Yaskawa INFORM job: DPRINT3D13.JBI

/JOB
//NAME DPRINT3D13
//POS
///NPOS 947,0,0,0,0,0
///TOOL 9
///POSTYPE PULSE
///PULSE
C00000=36504,50728,-112236,78231,-119117,-87318,0
C00001=42210,46378,-124713,70675,-118736,-91580,0
C00002=39842,45351,-127762,72820,-116851,-92177,0
C00003=34258,49660,-115138,80114,-117255,-87892,0
C00004=35160,50071,-114017,79347,-117985,-87668,0
C00005=34925,50304,-113369,79663,-117991,-87456,0
C00006=35393,50528,-112763,79272,-118380,-87336,0
C00007=35576,50347,-113263,79025,-118376,-87500,0
C00008=36136,50038,-114124,78353,-118497,-87812,0
C00009=41210,45662,-126843,71472,-117684,-92067,0
C00010=42439,44983,-128954,69897,-117543,-92821,0
C00011=39332,48664,-118025,74580,-119242,-89315,0
C00012=41658,49917,-114566,72665,-121338,-88655,0
C00013=34878,50571,-112636,79801,-118117,-87241,0
C00014=33997,51512,-110060,80995,-118129,-86405,0
C00015=36100,49514,-115576,78205,-118155,-88224,0
C00016=40170,46391,-124628,72850,-117873,-91306,0
C00017=40171,46330,-124643,72860,-117898,-91281,0
C00018=33600,46215,-124852,79721,-114877,-90646,0
C00019=36393,47272,-121802,77159,-116891,-90027,0
C00020=36323,49924,-114301,78154,-118581,-87857,0
C00021=40982,46356,-124583,72010,-118271,-91361,0
C00022=39975,45915,-125877,72916,-117468,-91614,0
C00023=35360,49470,-115543,78969,-117787,-88102,0
C00024=36245,49887,-114404,78220,-118516,-87877,0
C00025=35630,50238,-113425,78963,-118392,-87525,0
C00026=36504,50672,-112251,78242,-119134,-87295,0
C00027=42210,46316,-124729,70686,-118763,-91556,0
C00028=39843,45287,-127778,72830,-116876,-92151,0
C00029=34259,49603,-115155,80124,-117272,-87868,0
C00030=35161,50014,-114032,79357,-118002,-87645,0
C00031=34925,50248,-113384,79673,-118008,-87433,0
C00032=35394,50472,-112778,79282,-118397,-87313,0
C00033=35576,50291,-113278,79035,-118393,-87477,0
C00034=36137,49982,-114139,78363,-118516,-87789,0
C00035=41210,45599,-126858,71483,-117710,-92041,0
C00036=42421,44928,-128939,69931,-117572,-92784,0
C00037=39332,48606,-118041,74591,-119264,-89291,0
C00038=41626,49842,-114632,72703,-121329,-88642,0
C00039=34879,50515,-112651,79811,-118134,-87218,0
C00040=34010,51443,-110113,80987,-118144,-86395,0
C00041=36100,49457,-115591,78215,-118173,-88200,0
C00042=40171,46330,-124643,72860,-117898,-91281,0
C00043=40171,46268,-124659,72871,-117922,-91256,0
C00044=33640,46167,-124827,79692,-114924,-90612,0
C00045=36394,47211,-121817,77168,-116912,-90002,0
C00046=36324,49868,-114316,78165,-118600,-87834,0
C00047=40982,46294,-124599,72020,-118295,-91336,0
C00048=39976,45852,-125893,72926,-117492,-91589,0
C00049=35360,49413,-115558,78979,-117805,-88078,0
C00050=36246,49830,-114419,78230,-118534,-87854,0
C00051=35631,50182,-113440,78973,-118409,-87502,0
C00052=36504,50617,-112266,78252,-119152,-87272,0
C00053=42211,46254,-124744,70697,-118789,-91531,0
C00054=39843,45223,-127794,72840,-116901,-92125,0
C00055=34259,49546,-115170,80133,-117290,-87845,0
C00056=35161,49958,-114047,79366,-118019,-87622,0
C00057=34926,50192,-113399,79682,-118025,-87410,0
C00058=35394,50417,-112793,79292,-118415,-87290,0
C00059=35577,50235,-113293,79045,-118410,-87454,0
C00060=36137,49925,-114154,78373,-118533,-87765,0
C00061=41211,45536,-126874,71493,-117736,-92016,0
C00062=42403,44874,-128924,69965,-117602,-92748,0
C00063=39333,48548,-118056,74602,-119286,-89268,0
C00064=41594,49766,-114699,72740,-121321,-88629,0
C00065=34879,50459,-112666,79821,-118152,-87195,0
C00066=34023,51374,-110166,80980,-118160,-86384,0
C00067=36101,49400,-115607,78225,-118192,-88177,0
C00068=40171,46268,-124659,72871,-117922,-91256,0
C00069=40172,46206,-124674,72881,-117946,-91231,0
C00070=33681,46119,-124803,79663,-114971,-90578,0
C00071=36394,47151,-121832,77178,-116932,-89977,0
C00072=36324,49811,-114331,78175,-118618,-87811,0
C00073=40982,46232,-124614,72031,-118321,-91312,0
C00074=39976,45790,-125908,72937,-117517,-91563,0
C00075=35361,49356,-115573,78988,-117823,-88054,0
C00076=36246,49773,-114434,78240,-118553,-87830,0
C00077=35631,50126,-113455,78983,-118427,-87479,0
C00078=36505,50561,-112281,78263,-119171,-87249,0
C00079=42211,46192,-124760,70708,-118815,-91506,0
C00080=39843,45159,-127810,72850,-116927,-92100,0
C00081=34259,49489,-115184,80143,-117307,-87821,0
C00082=35161,49901,-114062,79376,-118037,-87599,0
C00083=34926,50136,-113414,79692,-118042,-87386,0
C00084=35394,50361,-112807,79302,-118432,-87267,0
C00085=35577,50179,-113308,79056,-118429,-87431,0
C00086=36137,49869,-114169,78383,-118551,-87742,0
C00087=41211,45472,-126890,71503,-117762,-91991,0
C00088=42385,44819,-128910,69999,-117632,-92711,0
C00089=39333,48489,-118071,74612,-119308,-89244,0
C00090=41562,49691,-114766,72778,-121312,-88616,0
C00091=34879,50404,-112681,79830,-118168,-87172,0
C00092=34036,51306,-110219,80972,-118176,-86374,0
C00093=36101,49343,-115622,78235,-118210,-88153,0
C00094=40172,46206,-124674,72881,-117946,-91231,0
C00095=40172,46144,-124690,72892,-117970,-91206,0
C00096=33721,46071,-124778,79635,-115017,-90544,0
C00097=36394,47091,-121848,77188,-116953,-89953,0
C00098=36324,49755,-114346,78185,-118637,-87787,0
C00099=40983,46170,-124631,72041,-118346,-91287,0
C00100=39976,45727,-125924,72947,-117541,-91538,0
C00101=35361,49299,-115588,78998,-117841,-88031,0
C00102=36246,49717,-114449,78250,-118571,-87807,0
C00103=35631,50070,-113469,78993,-118445,-87456,0
C00104=36505,50505,-112296,78273,-119188,-87226,0
C00105=42212,46130,-124775,70718,-118841,-91482,0
C00106=39844,45095,-127825,72860,-116952,-92074,0
C00107=34260,49432,-115199,80152,-117324,-87797,0
C00108=35161,49845,-114077,79386,-118054,-87576,0
C00109=34926,50080,-113429,79702,-118060,-87363,0
C00110=35395,50305,-112822,79312,-118449,-87244,0
C00111=35577,50123,-113323,79066,-118446,-87408,0
C00112=36138,49813,-114184,78394,-118570,-87719,0
C00113=41212,45409,-126905,71514,-117787,-91966,0
C00114=42367,44764,-128895,70033,-117662,-92674,0
C00115=39333,48431,-118086,74623,-119328,-89220,0
C00116=41530,49615,-114832,72816,-121304,-88603,0
C00117=34880,50348,-112696,79840,-118185,-87149,0
C00118=34049,51237,-110272,80965,-118192,-86364,0
C00119=36101,49286,-115637,78245,-118230,-88129,0
C00120=40172,46144,-124690,72892,-117970,-91206,0
C00121=40173,46082,-124705,72902,-117995,-91181,0
C00122=33761,46023,-124752,79606,-115064,-90509,0
C00123=36395,47031,-121863,77198,-116974,-89928,0
C00124=36325,49699,-114361,78195,-118655,-87764,0
C00125=40983,46108,-124645,72052,-118370,-91262,0
C00126=39977,45665,-125939,72957,-117567,-91513,0
C00127=35361,49242,-115603,79008,-117859,-88007,0
C00128=36247,49661,-114464,78260,-118589,-87784,0
C00129=35632,50014,-113484,79003,-118462,-87433,0
C00130=36505,50450,-112310,78283,-119207,-87203,0
C00131=42212,46068,-124791,70729,-118866,-91457,0
C00132=39844,45031,-127841,72870,-116977,-92048,0
C00133=34260,49376,-115213,80162,-117341,-87773,0
C00134=35162,49789,-114092,79396,-118072,-87552,0
C00135=34927,50024,-113444,79712,-118077,-87340,0
C00136=35395,50249,-112837,79322,-118466,-87220,0
C00137=35578,50067,-113337,79076,-118463,-87385,0
C00138=36138,49756,-114199,78404,-118588,-87696,0
C00139=41212,45346,-126921,71524,-117814,-91940,0
C00140=42349,44709,-128880,70067,-117692,-92638,0
C00141=39334,48373,-118101,74634,-119350,-89196,0
C00142=41497,49539,-114898,72854,-121295,-88589,0
C00143=34880,50292,-112711,79850,-118202,-87125,0
C00144=34062,51168,-110325,80957,-118207,-86354,0
C00145=36102,49229,-115651,78255,-118248,-88106,0
C00146=40173,46082,-124705,72902,-117995,-91181,0
C00147=40173,46020,-124720,72913,-118019,-91156,0
C00148=33801,45976,-124727,79578,-115111,-90475,0
C00149=36395,46971,-121878,77207,-116993,-89903,0
C00150=36325,49642,-114375,78206,-118673,-87740,0
C00151=40984,46047,-124660,72063,-118395,-91237,0
C00152=39977,45602,-125955,72967,-117591,-91488,0
C00153=35362,49185,-115618,79018,-117877,-87984,0
C00154=36247,49604,-114478,78271,-118608,-87761,0
C00155=35632,49958,-113499,79013,-118480,-87410,0
C00156=36506,50394,-112325,78294,-119224,-87180,0
C00157=42212,46006,-124806,70740,-118893,-91433,0
C00158=39845,44968,-127856,72880,-117002,-92022,0
C00159=34260,49319,-115228,80171,-117359,-87750,0
C00160=35162,49733,-114106,79406,-118090,-87529,0
C00161=34927,49968,-113458,79722,-118093,-87317,0
C00162=35395,50194,-112851,79332,-118484,-87197,0
C00163=35578,50011,-113352,79086,-118481,-87361,0
C00164=36138,49700,-114214,78414,-118607,-87672,0
C00165=41213,45283,-126936,71535,-117840,-91915,0
C00166=42331,44655,-128865,70101,-117721,-92601,0
C00167=39334,48315,-118116,74645,-119372,-89172,0
C00168=41465,49464,-114964,72892,-121286,-88577,0
C00169=34880,50237,-112725,79860,-118218,-87102,0
C00170=34075,51099,-110378,80950,-118223,-86343,0
C00171=36102,49172,-115666,78265,-118266,-88082,0
C00172=40173,46020,-124720,72913,-118019,-91156,0
C00173=40173,45959,-124736,72923,-118044,-91131,0
C00174=33841,45928,-124702,79550,-115157,-90441,0
C00175=36396,46910,-121893,77217,-117014,-89878,0
C00176=36325,49586,-114390,78216,-118692,-87717,0
C00177=40984,45985,-124676,72074,-118420,-91212,0
C00178=39978,45540,-125970,72978,-117615,-91462,0
C00179=35362,49128,-115633,79028,-117895,-87960,0
C00180=36247,49548,-114493,78281,-118626,-87737,0
C00181=35632,49902,-113513,79023,-118497,-87386,0
C00182=36506,50339,-112339,78304,-119242,-87157,0
C00183=42213,45944,-124821,70751,-118918,-91408,0
C00184=39845,44904,-127872,72890,-117028,-91997,0
C00185=34261,49262,-115243,80181,-117376,-87726,0
C00186=35163,49676,-114121,79416,-118107,-87505,0
C00187=34927,49912,-113473,79732,-118110,-87294,0
C00188=35396,50138,-112866,79342,-118501,-87175,0
C00189=35578,49955,-113367,79096,-118499,-87338,0
C00190=36139,49644,-114228,78424,-118624,-87649,0
C00191=41213,45220,-126952,71545,-117865,-91890,0
C00192=42313,44600,-128849,70135,-117751,-92565,0
C00193=39334,48257,-118131,74656,-119394,-89149,0
C00194=41433,49388,-115030,72930,-121277,-88563,0
C00195=34881,50181,-112740,79870,-118235,-87079,0
C00196=34088,51030,-110431,80942,-118239,-86332,0
C00197=36102,49115,-115681,78276,-118285,-88058,0
C00198=40173,45959,-124736,72923,-118044,-91131,0
C00199=40174,45897,-124751,72934,-118068,-91106,0
C00200=33881,45880,-124675,79522,-115204,-90407,0
C00201=36396,46850,-121908,77227,-117035,-89853,0
C00202=36326,49529,-114404,78226,-118710,-87693,0
C00203=40984,45923,-124691,72084,-118446,-91187,0
C00204=39978,45477,-125985,72988,-117640,-91437,0
C00205=35362,49071,-115646,79038,-117913,-87936,0
C00206=36248,49491,-114507,78291,-118645,-87714,0
C00207=35633,49846,-113528,79033,-118515,-87363,0
C00208=36506,50284,-112354,78315,-119261,-87135,0
C00209=42213,45883,-124836,70762,-118944,-91383,0
C00210=39846,44840,-127887,72900,-117053,-91971,0
C00211=34261,49205,-115258,80190,-117393,-87702,0
C00212=35163,49620,-114136,79426,-118124,-87482,0
C00213=34928,49856,-113487,79742,-118127,-87270,0
C00214=35396,50082,-112880,79352,-118519,-87151,0
C00215=35579,49899,-113381,79106,-118516,-87314,0
C00216=36139,49587,-114243,78435,-118642,-87625,0
C00217=41213,45157,-126967,71556,-117892,-91864,0
C00218=42295,44546,-128834,70169,-117780,-92528,0
C00219=39335,48198,-118145,74667,-119414,-89125,0
C00220=41400,49313,-115096,72967,-121269,-88550,0
C00221=34881,50125,-112754,79880,-118253,-87056,0
C00222=34101,50961,-110484,80935,-118255,-86322,0
C00223=36103,49058,-115696,78286,-118303,-88035,0
C00224=40174,45897,-124751,72934,-118068,-91106,0
C00225=40174,45835,-124766,72944,-118092,-91081,0
C00226=33921,45833,-124650,79494,-115251,-90372,0
C00227=36396,46790,-121923,77237,-117055,-89828,0
C00228=36326,49473,-114419,78237,-118728,-87670,0
C00229=40985,45861,-124706,72095,-118470,-91162,0
C00230=39978,45415,-126000,72998,-117664,-91411,0
C00231=35363,49014,-115661,79048,-117931,-87912,0
C00232=36248,49435,-114522,78302,-118663,-87690,0
C00233=35633,49790,-113542,79044,-118533,-87339,0
C00234=36507,50228,-112368,78326,-119278,-87111,0
C00235=42214,45821,-124851,70773,-118971,-91358,0
C00236=39846,44777,-127902,72910,-117078,-91945,0
C00237=34261,49149,-115272,80200,-117410,-87678,0
C00238=35163,49564,-114150,79436,-118142,-87458,0
C00239=34928,49800,-113502,79752,-118145,-87247,0
C00240=35396,50026,-112895,79362,-118537,-87128,0
C00241=35579,49843,-113395,79116,-118534,-87291,0
C00242=36139,49531,-114257,78445,-118661,-87602,0
C00243=41214,45093,-126982,71566,-117918,-91839,0
C00244=42277,44492,-128819,70203,-117810,-92492,0
C00245=39335,48140,-118160,74678,-119436,-89101,0
C00246=41368,49237,-115161,73006,-121260,-88537,0
C00247=34881,50070,-112768,79890,-118270,-87032,0
C00248=34114,50893,-110536,80927,-118271,-86311,0
C00249=36103,49001,-115710,78296,-118322,-88011,0
C00250=40174,45835,-124766,72944,-118092,-91081,0
C00251=40175,45773,-124781,72955,-118117,-91055,0
C00252=33961,45785,-124624,79466,-115298,-90338,0
C00253=36397,46730,-121938,77246,-117076,-89803,0
C00254=36326,49417,-114433,78247,-118747,-87647,0
C00255=40985,45800,-124721,72106,-118495,-91137,0
C00256=39979,45352,-126015,73009,-117690,-91386,0
C00257=35363,48957,-115675,79058,-117949,-87888,0
C00258=36248,49379,-114536,78312,-118681,-87667,0
C00259=35633,49734,-113556,79054,-118550,-87316,0
C00260=36507,50173,-112382,78336,-119296,-87088,0
C00261=42214,45759,-124866,70784,-118996,-91333,0
C00262=39846,44713,-127918,72921,-117104,-91919,0
C00263=34262,49092,-115287,80210,-117426,-87655,0
C00264=35163,49508,-114164,79446,-118160,-87435,0
C00265=34928,49744,-113516,79762,-118162,-87223,0
C00266=35397,49971,-112909,79373,-118554,-87104,0
C00267=35579,49788,-113410,79127,-118551,-87268,0
C00268=36140,49475,-114271,78455,-118679,-87578,0
C00269=41214,45030,-126997,71577,-117944,-91814,0
C00270=42259,44437,-128803,70237,-117840,-92455,0
C00271=39336,48082,-118175,74689,-119458,-89077,0
C00272=41336,49162,-115227,73044,-121252,-88523,0
C00273=34882,50014,-112783,79900,-118287,-87009,0
C00274=34127,50824,-110589,80920,-118287,-86300,0
C00275=36103,48944,-115725,78306,-118340,-87988,0
C00276=40175,45773,-124781,72955,-118117,-91055,0
C00277=40175,45712,-124796,72965,-118141,-91030,0
C00278=34001,45738,-124598,79438,-115345,-90304,0
C00279=36397,46670,-121952,77256,-117097,-89778,0
C00280=36327,49360,-114447,78257,-118765,-87623,0
C00281=40986,45738,-124736,72117,-118520,-91112,0
C00282=39979,45290,-126030,73019,-117715,-91361,0
C00283=35363,48900,-115690,79068,-117968,-87865,0
C00284=36249,49322,-114550,78322,-118700,-87643,0
C00285=35634,49678,-113571,79064,-118569,-87292,0
C00286=36507,50117,-112397,78347,-119315,-87065,0
C00287=42215,45697,-124881,70795,-119023,-91308,0
C00288=39847,44649,-127933,72931,-117129,-91893,0
C00289=34262,49035,-115301,80219,-117444,-87631,0
C00290=35164,49452,-114178,79456,-118177,-87411,0
C00291=34929,49688,-113530,79772,-118179,-87200,0
C00292=35397,49915,-112923,79383,-118571,-87081,0
C00293=35580,49732,-113424,79137,-118569,-87245,0
C00294=36140,49419,-114286,78466,-118697,-87555,0
C00295=41215,44967,-127012,71587,-117970,-91788,0
C00296=42241,44383,-128788,70271,-117869,-92418,0
C00297=39336,48024,-118188,74700,-119480,-89054,0
C00298=41303,49086,-115292,73082,-121243,-88509,0
C00299=34882,49959,-112797,79910,-118303,-86986,0
C00300=34140,50755,-110641,80913,-118303,-86290,0
C00301=36104,48888,-115738,78316,-118360,-87964,0
C00302=40175,45712,-124796,72965,-118141,-91030,0
C00303=40175,45650,-124811,72976,-118165,-91005,0
C00304=34041,45691,-124572,79410,-115392,-90269,0
C00305=36397,46610,-121967,77266,-117117,-89753,0
C00306=36327,49304,-114462,78268,-118784,-87599,0
C00307=40986,45676,-124750,72128,-118546,-91087,0
C00308=39980,45227,-126045,73030,-117739,-91335,0
C00309=35364,48844,-115704,79078,-117985,-87841,0
C00310=36249,49266,-114565,78333,-118718,-87620,0
C00311=35634,49622,-113585,79074,-118586,-87269,0
C00312=36508,50062,-112411,78357,-119332,-87042,0
C00313=42215,45636,-124896,70807,-119049,-91283,0
C00314=39847,44586,-127948,72941,-117154,-91867,0
C00315=34262,48979,-115314,80229,-117461,-87607,0
C00316=35164,49396,-114193,79466,-118194,-87388,0
C00317=34929,49633,-113544,79782,-118196,-87176,0
C00318=35397,49860,-112937,79393,-118588,-87058,0
C00319=35580,49676,-113438,79147,-118587,-87221,0
C00320=36140,49362,-114300,78476,-118716,-87531,0
C00321=41215,44904,-127027,71598,-117996,-91763,0
C00322=42223,44329,-128772,70305,-117899,-92381,0
C00323=39336,47966,-118203,74711,-119502,-89030,0
C00324=41271,49010,-115358,73120,-121235,-88496,0
C00325=34882,49903,-112811,79920,-118321,-86963,0
C00326=34153,50686,-110693,80905,-118319,-86279,0
C00327=36104,48831,-115752,78327,-118378,-87940,0
C00328=40175,45650,-124811,72976,-118165,-91005,0
C00329=40176,45588,-124825,72987,-118191,-90980,0
C00330=34081,45644,-124545,79383,-115440,-90235,0
C00331=36398,46550,-121982,77276,-117138,-89728,0
C00332=36327,49248,-114476,78278,-118802,-87576,0
C00333=40987,45615,-124765,72138,-118571,-91062,0
C00334=39980,45165,-126060,73040,-117764,-91310,0
C00335=35364,48787,-115719,79088,-118003,-87817,0
C00336=36249,49210,-114579,78343,-118736,-87596,0
C00337=35634,49566,-113599,79085,-118604,-87245,0
C00338=36508,50007,-112425,78368,-119350,-87019,0
C00339=42215,45574,-124911,70818,-119075,-91259,0
C00340=39848,44522,-127963,72951,-117179,-91841,0
C00341=34263,48922,-115329,80239,-117478,-87583,0
C00342=35164,49339,-114207,79476,-118212,-87364,0
C00343=34929,49577,-113558,79792,-118214,-87153,0
C00344=35398,49804,-112951,79403,-118605,-87035,0
C00345=35580,49620,-113452,79157,-118604,-87198,0
C00346=36141,49306,-114314,78487,-118734,-87508,0
C00347=41215,44841,-127041,71609,-118022,-91737,0
C00348=42205,44275,-128756,70339,-117929,-92345,0
C00349=39337,47908,-118217,74722,-119523,-89005,0
C00350=41238,48935,-115423,73158,-121226,-88482,0
C00351=34883,49848,-112825,79930,-118338,-86939,0
C00352=34166,50617,-110745,80898,-118335,-86268,0
C00353=36104,48774,-115767,78337,-118396,-87916,0
C00354=40176,45588,-124825,72987,-118191,-90980,0
C00355=40176,45527,-124840,72997,-118215,-90954,0
C00356=34121,45597,-124519,79355,-115488,-90201,0
C00357=36398,46490,-121996,77286,-117159,-89702,0
C00358=36328,49192,-114490,78289,-118820,-87552,0
C00359=40987,45553,-124780,72149,-118596,-91037,0
C00360=39981,45102,-126075,73051,-117788,-91283,0
C00361=35364,48730,-115733,79098,-118022,-87793,0
C00362=36250,49153,-114593,78354,-118755,-87572,0
C00363=35635,49511,-113613,79095,-118622,-87222,0
C00364=36508,49951,-112439,78379,-119369,-86995,0
C00365=42216,45512,-124925,70829,-119101,-91234,0
C00366=39848,44458,-127978,72962,-117205,-91815,0
C00367=34263,48865,-115343,80249,-117495,-87559,0
C00368=35165,49283,-114221,79486,-118230,-87340,0
C00369=34929,49521,-113572,79802,-118231,-87129,0
C00370=35398,49749,-112965,79414,-118623,-87011,0
C00371=35581,49564,-113466,79168,-118622,-87174,0
C00372=36141,49250,-114328,78497,-118753,-87484,0
C00373=41216,44778,-127056,71620,-118048,-91711,0
C00374=42188,44221,-128741,70374,-117957,-92308,0
C00375=39337,47850,-118231,74733,-119544,-88982,0
C00376=41206,48859,-115489,73196,-121218,-88469,0
C00377=34883,49792,-112839,79940,-118355,-86916,0
C00378=34179,50549,-110798,80891,-118352,-86257,0
C00379=36105,48717,-115781,78347,-118415,-87892,0
C00380=40176,45527,-124840,72997,-118215,-90954,0
C00381=40177,45465,-124855,73008,-118239,-90930,0
C00382=34161,45550,-124493,79328,-115535,-90166,0
C00383=36398,46430,-122009,77296,-117179,-89677,0
C00384=36328,49136,-114503,78299,-118839,-87529,0
C00385=40987,45492,-124794,72160,-118622,-91012,0
C00386=39981,45040,-126089,73061,-117814,-91258,0
C00387=35365,48673,-115746,79108,-118040,-87769,0
C00388=36250,49097,-114607,78364,-118773,-87549,0
C00389=35635,49455,-113627,79105,-118639,-87198,0
C00390=36509,49896,-112452,78390,-119387,-86972,0
C00391=42216,45451,-124940,70840,-119127,-91209,0
C00392=39848,44395,-127993,72972,-117230,-91789,0
C00393=34263,48809,-115357,80258,-117513,-87535,0
C00394=35165,49227,-114235,79497,-118247,-87316,0
C00395=34930,49465,-113586,79812,-118248,-87106,0
C00396=35398,49693,-112979,79424,-118641,-86988,0
C00397=35581,49509,-113480,79178,-118640,-87151,0
C00398=36141,49194,-114342,78507,-118771,-87461,0
C00399=41216,44715,-127071,71630,-118075,-91686,0
C00400=42170,44167,-128725,70408,-117987,-92271,0
C00401=39337,47792,-118246,74745,-119566,-88958,0
C00402=41173,48784,-115553,73235,-121209,-88455,0
C00403=34883,49737,-112853,79951,-118372,-86892,0
C00404=34192,50480,-110849,80883,-118368,-86246,0
C00405=36105,48660,-115795,78358,-118434,-87868,0
C00406=40177,45465,-124855,73008,-118239,-90930,0
C00407=40177,45404,-124868,73019,-118264,-90904,0
C00408=34200,45503,-124465,79301,-115582,-90132,0
C00409=36399,46370,-122024,77306,-117200,-89652,0
C00410=36328,49080,-114517,78310,-118857,-87505,0
C00411=40988,45430,-124809,72171,-118646,-90987,0
C00412=39981,44978,-126104,73072,-117839,-91232,0
C00413=35365,48616,-115760,79118,-118057,-87745,0
C00414=36250,49041,-114620,78375,-118792,-87525,0
C00415=35635,49399,-113640,79116,-118657,-87175,0
C00416=36509,49841,-112466,78400,-119404,-86949,0
C00417=42217,45389,-124955,70852,-119154,-91184,0
C00418=39849,44331,-128007,72982,-117255,-91763,0
C00419=34264,48752,-115371,80268,-117530,-87511,0
C00420=35165,49171,-114248,79507,-118265,-87292,0
C00421=34930,49409,-113600,79822,-118265,-87082,0
C00422=35399,49638,-112993,79434,-118658,-86965,0
C00423=35581,49453,-113494,79188,-118657,-87127,0
C00424=36142,49138,-114356,78518,-118788,-87437,0
C00425=41217,44652,-127085,71641,-118101,-91660,0
C00426=42152,44113,-128709,70442,-118017,-92234,0
C00427=39338,47734,-118260,74756,-119588,-88933,0
C00428=41140,48708,-115619,73273,-121200,-88441,0
C00429=34883,49681,-112867,79961,-118389,-86869,0
C00430=34205,50411,-110901,80876,-118384,-86236,0
C00431=36105,48604,-115808,78368,-118453,-87844,0
C00432=40177,45404,-124868,73019,-118264,-90904,0
C00433=40177,45342,-124883,73030,-118288,-90878,0
C00434=34240,45456,-124439,79274,-115630,-90098,0
C00435=36399,46310,-122038,77316,-117221,-89627,0
C00436=36329,49023,-114531,78321,-118876,-87482,0
C00437=40988,45369,-124822,72182,-118671,-90961,0
C00438=39982,44915,-126119,73083,-117863,-91207,0
C00439=35365,48560,-115774,79129,-118076,-87721,0
C00440=36251,48985,-114634,78385,-118810,-87501,0
C00441=35636,49343,-113654,79126,-118674,-87151,0
C00442=36509,49786,-112480,78411,-119423,-86926,0
C00443=42217,45327,-124968,70863,-119180,-91159,0
C00444=39849,44268,-128022,72993,-117282,-91736,0
C00445=34264,48696,-115384,80278,-117548,-87487,0
C00446=35166,49115,-114262,79517,-118283,-87269,0
C00447=34930,49354,-113614,79832,-118284,-87058,0
C00448=35399,49582,-113007,79445,-118676,-86941,0
C00449=35582,49397,-113507,79199,-118676,-87104,0
C00450=36142,49082,-114369,78528,-118807,-87414,0
C00451=41217,44589,-127100,71652,-118127,-91635,0
C00452=42134,44059,-128693,70476,-118046,-92197,0
C00453=39338,47676,-118273,74767,-119610,-88910,0
C00454=41108,48633,-115683,73312,-121192,-88427,0
C00455=34884,49626,-112880,79971,-118406,-86845,0
C00456=34218,50342,-110953,80869,-118401,-86225,0
C00457=36106,48547,-115822,78379,-118471,-87820,0
C00458=40177,45342,-124883,73030,-118288,-90878,0
C00459=40178,45280,-124897,73041,-118314,-90854,0
C00460=34280,45409,-124411,79247,-115677,-90064,0
C00461=36400,46250,-122052,77326,-117241,-89601,0
C00462=36329,48967,-114545,78331,-118895,-87458,0
C00463=40989,45307,-124837,72194,-118696,-90936,0
C00464=39982,44853,-126132,73093,-117888,-91181,0
C00465=35366,48503,-115788,79139,-118094,-87697,0
C00466=36251,48929,-114648,78396,-118828,-87478,0
C00467=35636,49288,-113668,79137,-118693,-87128,0
C00468=36509,49730,-112494,78422,-119441,-86902,0
C00469=42217,45266,-124982,70874,-119207,-91134,0
C00470=39850,44204,-128037,73003,-117307,-91710,0
C00471=34264,48639,-115398,80288,-117566,-87463,0
C00472=35166,49059,-114276,79527,-118300,-87245,0
C00473=34931,49298,-113627,79843,-118301,-87035,0
C00474=35399,49527,-113020,79455,-118693,-86918,0
C00475=35582,49342,-113521,79209,-118693,-87080,0
C00476=36142,49026,-114383,78539,-118825,-87390,0
C00477=41218,44526,-127115,71663,-118154,-91608,0
C00478=42116,44005,-128676,70511,-118076,-92160,0
C00479=39338,47618,-118287,74778,-119632,-88885,0
C00480=41075,48557,-115748,73350,-121184,-88413,0
C00481=34884,49571,-112894,79981,-118423,-86822,0
C00482=34232,50273,-111005,80861,-118417,-86214,0
C00483=36106,48490,-115836,78389,-118489,-87796,0
C00484=40178,45280,-124897,73041,-118314,-90854,0
C00485=40178,45219,-124911,73052,-118338,-90828,0
C00486=34319,45363,-124385,79220,-115725,-90029,0
C00487=36400,46190,-122066,77336,-117262,-89576,0
C00488=36329,48911,-114558,78342,-118913,-87434,0
C00489=40989,45246,-124851,72205,-118722,-90911,0
C00490=39983,44791,-126146,73104,-117914,-91155,0
C00491=35366,48446,-115802,79149,-118113,-87672,0
C00492=36251,48873,-114661,78407,-118847,-87454,0
C00493=35636,49232,-113681,79147,-118710,-87104,0
C00494=36510,49675,-112507,78433,-119459,-86879,0
C00495=42218,45204,-124997,70886,-119232,-91109,0
C00496=39850,44141,-128050,73014,-117332,-91684,0
C00497=34265,48583,-115412,80298,-117583,-87439,0
C00498=35166,49003,-114289,79537,-118318,-87222,0
C00499=34931,49242,-113641,79853,-118318,-87011,0
C00500=35400,49471,-113034,79465,-118710,-86894,0
C00501=35582,49286,-113535,79220,-118711,-87056,0
C00502=36143,48970,-114397,78550,-118843,-87366,0
C00503=41218,44464,-127129,71674,-118179,-91583,0
C00504=42098,43952,-128659,70545,-118104,-92124,0
C00505=39339,47560,-118301,74790,-119654,-88861,0
C00506=41042,48482,-115812,73389,-121175,-88399,0
C00507=34884,49515,-112908,79991,-118440,-86798,0
C00508=34245,50205,-111057,80854,-118433,-86203,0
C00509=36106,48433,-115850,78400,-118509,-87772,0
C00510=40178,45219,-124911,73052,-118338,-90828,0
C00511=40179,45157,-124925,73063,-118362,-90802,0
C00512=34359,45316,-124357,79193,-115773,-89995,0
C00513=36400,46131,-122081,77346,-117283,-89551,0
C00514=36330,48855,-114572,78353,-118932,-87410,0
C00515=40989,45184,-124865,72216,-118747,-90886,0
C00516=39983,44729,-126161,73115,-117938,-91130,0
C00517=35366,48390,-115815,79159,-118131,-87649,0
C00518=36252,48816,-114675,78417,-118865,-87430,0
C00519=35637,49176,-113695,79158,-118728,-87081,0
C00520=36510,49620,-112520,78444,-119477,-86855,0
C00521=42218,45143,-125011,70897,-119258,-91083,0
C00522=39851,44077,-128065,73024,-117358,-91658,0
C00523=34265,48526,-115426,80308,-117600,-87415,0
C00524=35167,48947,-114303,79548,-118335,-87197,0
C00525=34931,49187,-113654,79863,-118335,-86987,0
C00526=35400,49416,-113047,79476,-118728,-86870,0
C00527=35583,49230,-113548,79230,-118728,-87033,0
C00528=36143,48914,-114410,78560,-118862,-87342,0
C00529=41218,44401,-127143,71685,-118206,-91557,0
C00530=42081,43898,-128643,70579,-118134,-92087,0
C00531=39339,47503,-118315,74801,-119675,-88837,0
C00532=41010,48406,-115876,73427,-121167,-88384,0
C00533=34885,49460,-112921,80002,-118457,-86775,0
C00534=34258,50136,-111108,80847,-118449,-86192,0
C00535=36107,48377,-115864,78410,-118527,-87748,0
C00536=40179,45157,-124925,73063,-118362,-90802,0
C00537=40179,45096,-124940,73073,-118387,-90777,0
C00538=34399,45270,-124329,79166,-115821,-89960,0
C00539=36401,46071,-122094,77357,-117304,-89525,0
C00540=36330,48799,-114585,78363,-118950,-87386,0
C00541=40990,45123,-124880,72227,-118772,-90860,0
C00542=39983,44666,-126175,73125,-117963,-91104,0
C00543=35367,48333,-115828,79169,-118149,-87624,0
C00544=36252,48760,-114688,78428,-118885,-87406,0
C00545=35637,49121,-113708,79168,-118747,-87057,0
C00546=36511,49565,-112534,78454,-119495,-86832,0
C00547=42219,45081,-125025,70908,-119285,-91058,0
C00548=39851,44014,-128079,73035,-117384,-91631,0
C00549=34265,48470,-115438,80317,-117617,-87390,0
C00550=35167,48891,-114316,79558,-118353,-87173,0
C00551=34932,49131,-113668,79873,-118353,-86963,0
C00552=35400,49361,-113061,79486,-118746,-86847,0
C00553=35583,49175,-113562,79241,-118746,-87009,0
C00554=36143,48858,-114423,78571,-118880,-87319,0
C00555=41219,44338,-127158,71696,-118232,-91531,0
C00556=42063,43845,-128626,70613,-118163,-92049,0
C00557=39340,47445,-118329,74812,-119697,-88813,0
C00558=40977,48330,-115941,73466,-121159,-88371,0
C00559=34885,49405,-112934,80012,-118474,-86751,0
C00560=34271,50067,-111160,80840,-118466,-86180,0
C00561=36107,48320,-115877,78421,-118546,-87724,0
C00562=40179,45096,-124940,73073,-118387,-90777,0
C00563=40179,45034,-124953,73084,-118411,-90751,0
C00564=34438,45223,-124302,79140,-115868,-89926,0
C00565=36401,46011,-122107,77367,-117324,-89500,0
C00566=36330,48743,-114599,78374,-118969,-87363,0
C00567=40990,45061,-124894,72238,-118797,-90835,0
C00568=39984,44604,-126189,73136,-117988,-91078,0
C00569=35367,48277,-115842,79180,-118167,-87600,0
C00570=36252,48704,-114702,78438,-118903,-87382,0
C00571=35637,49065,-113722,79179,-118764,-87033,0
C00572=36511,49510,-112547,78465,-119513,-86809,0
C00573=42219,45020,-125038,70920,-119311,-91033,0
C00574=39851,43950,-128093,73045,-117409,-91605,0
C00575=34266,48413,-115452,80327,-117634,-87366,0
C00576=35167,48835,-114330,79568,-118371,-87150,0
C00577=34932,49076,-113681,79884,-118370,-86940,0
C00578=35400,49305,-113074,79497,-118763,-86823,0
C00579=35583,49119,-113575,79251,-118764,-86985,0
C00580=36144,48802,-114437,78582,-118899,-87295,0
C00581=41219,44275,-127171,71707,-118258,-91505,0
C00582=42045,43791,-128610,70648,-118192,-92012,0
C00583=39340,47387,-118341,74824,-119719,-88789,0
C00584=40944,48255,-116005,73505,-121150,-88356,0
C00585=34885,49349,-112948,80022,-118492,-86727,0
C00586=34284,49998,-111211,80833,-118483,-86169,0
C00587=36107,48263,-115890,78431,-118565,-87700,0
C00588=40179,45034,-124953,73084,-118411,-90751,0
C00589=40180,44973,-124967,73095,-118437,-90726,0
C00590=34478,45177,-124274,79113,-115916,-89892,0
C00591=36401,45951,-122121,77377,-117345,-89475,0
C00592=36331,48687,-114612,78385,-118987,-87339,0
C00593=40991,45000,-124907,72249,-118823,-90810,0
C00594=39984,44542,-126203,73147,-118013,-91052,0
C00595=35367,48220,-115856,79190,-118185,-87576,0
C00596=36253,48648,-114715,78449,-118922,-87359,0
C00597=35638,49009,-113735,79189,-118782,-87009,0
C00598=36511,49455,-112560,78476,-119532,-86785,0
C00599=42220,44958,-125052,70932,-119338,-91008,0
C00600=39852,43887,-128107,73056,-117435,-91579,0
C00601=34266,48357,-115466,80337,-117652,-87342,0
C00602=35168,48780,-114343,79579,-118388,-87126,0
C00603=34932,49020,-113694,79894,-118387,-86916,0
C00604=35401,49250,-113087,79507,-118780,-86799,0
C00605=35584,49064,-113588,79262,-118781,-86962,0
C00606=36144,48746,-114450,78592,-118917,-87271,0
C00607=41220,44212,-127185,71718,-118285,-91480,0
C00608=42027,43738,-128593,70682,-118222,-91976,0
C00609=39340,47329,-118355,74835,-119741,-88765,0
C00610=40911,48179,-116068,73544,-121142,-88342,0
C00611=34886,49294,-112961,80033,-118509,-86703,0
C00612=34297,49929,-111262,80825,-118500,-86158,0
C00613=36108,48207,-115904,78442,-118584,-87676,0
C00614=40180,44973,-124967,73095,-118437,-90726,0
C00615=40180,44912,-124981,73107,-118461,-90700,0
C00616=34517,45131,-124247,79087,-115965,-89857,0
C00617=36402,45891,-122135,77387,-117366,-89449,0
C00618=36331,48631,-114625,78396,-119005,-87315,0
C00619=40991,44938,-124921,72261,-118848,-90784,0
C00620=39985,44480,-126216,73158,-118038,-91026,0
C00621=35368,48163,-115868,79200,-118203,-87552,0
C00622=36253,48592,-114728,78460,-118940,-87334,0
C00623=35638,48954,-113748,79200,-118800,-86985,0
C00624=36512,49400,-112573,78487,-119550,-86762,0
C00625=42220,44897,-125066,70943,-119364,-90983,0
C00626=39852,43824,-128122,73066,-117460,-91552,0
C00627=34266,48301,-115479,80347,-117669,-87318,0
C00628=35168,48724,-114356,79589,-118407,-87102,0
C00629=34933,48964,-113707,79904,-118404,-86892,0
C00630=35401,49195,-113100,79518,-118799,-86775,0
C00631=35584,49008,-113601,79272,-118800,-86938,0
C00632=36144,48690,-114463,78603,-118935,-87247,0
C00633=41220,44149,-127199,71729,-118311,-91454,0
C00634=42009,43684,-128576,70717,-118250,-91939,0
C00635=39341,47271,-118369,74847,-119763,-88740,0
C00636=40878,48104,-116133,73582,-121134,-88328,0
C00637=34886,49239,-112974,80043,-118526,-86680,0
C00638=34311,49861,-111313,80818,-118516,-86146,0
C00639=36108,48150,-115916,78452,-118602,-87652,0
C00640=40180,44912,-124981,73107,-118461,-90700,0
C00641=40181,44850,-124995,73118,-118486,-90675,0
C00642=34557,45085,-124218,79061,-116013,-89823,0
C00643=36402,45832,-122148,77397,-117386,-89424,0
C00644=36331,48575,-114638,78406,-119025,-87291,0
C00645=40991,44877,-124934,72272,-118873,-90759,0
C00646=39985,44418,-126230,73169,-118063,-91000,0
C00647=35368,48107,-115882,79211,-118222,-87527,0
C00648=36253,48536,-114741,78471,-118958,-87310,0
C00649=35638,48898,-113761,79210,-118818,-86962,0
C00650=36512,49345,-112587,78498,-119567,-86738,0
C00651=42220,44835,-125080,70955,-119390,-90957,0
C00652=39853,43760,-128135,73077,-117486,-91525,0
C00653=34267,48244,-115491,80357,-117686,-87294,0
C00654=35168,48668,-114369,79600,-118424,-87078,0
C00655=34933,48909,-113721,79915,-118422,-86868,0
C00656=35402,49139,-113113,79528,-118816,-86752,0
C00657=35584,48953,-113614,79283,-118817,-86914,0
C00658=36145,48634,-114476,78614,-118955,-87223,0
C00659=41221,44087,-127213,71740,-118338,-91427,0
C00660=41992,43631,-128558,70751,-118279,-91901,0
C00661=39341,47214,-118381,74858,-119785,-88716,0
C00662=40846,48028,-116196,73621,-121126,-88313,0
C00663=34886,49184,-112987,80053,-118543,-86656,0
C00664=34324,49792,-111364,80811,-118533,-86135,0
C00665=36108,48094,-115930,78463,-118622,-87627,0
C00666=40181,44850,-124995,73118,-118486,-90675,0
C00667=40181,44789,-125007,73129,-118510,-90649,0
C00668=34596,45039,-124190,79035,-116061,-89789,0
C00669=36402,45772,-122161,77408,-117408,-89398,0
C00670=36332,48519,-114651,78417,-119043,-87267,0
C00671=40992,44816,-124948,72283,-118900,-90733,0
C00672=39985,44355,-126244,73180,-118088,-90974,0
C00673=35368,48050,-115895,79221,-118240,-87503,0
C00674=36254,48480,-114754,78481,-118977,-87287,0
C00675=35639,48843,-113774,79221,-118835,-86938,0
C00676=36512,49290,-112599,78509,-119586,-86715,0
C00677=42221,44774,-125094,70966,-119417,-90932,0
C00678=39853,43697,-128149,73088,-117511,-91499,0
C00679=34267,48188,-115505,80368,-117703,-87269,0
C00680=35169,48612,-114382,79610,-118442,-87054,0
C00681=34933,48853,-113734,79925,-118440,-86844,0
C00682=35402,49084,-113126,79539,-118833,-86728,0
C00683=35585,48897,-113627,79294,-118835,-86890,0
C00684=36145,48578,-114489,78624,-118973,-87199,0
C00685=39341,47156,-118395,74870,-119806,-88691,0
C00686=40813,47953,-116260,73660,-121116,-88299,0
C00687=36109,48037,-115943,78474,-118640,-87603,0
C00688=40181,44789,-125007,73129,-118510,-90649,0
C00689=40181,44728,-125021,73140,-118535,-90623,0
C00690=34635,44993,-124162,79009,-116110,-89754,0
C00691=36403,45712,-122175,77418,-117429,-89373,0
C00692=36332,48463,-114664,78428,-119062,-87243,0
C00693=40992,44754,-124961,72295,-118925,-90708,0
C00694=39986,44293,-126258,73191,-118114,-90948,0
C00695=35369,47994,-115907,79232,-118258,-87479,0
C00696=36254,48424,-114767,78492,-118996,-87262,0
C00697=35639,48787,-113787,79232,-118854,-86914,0
C00698=36512,49235,-112612,78520,-119604,-86691,0
C00699=42221,44712,-125107,70978,-119443,-90907,0
C00700=39853,43633,-128163,73098,-117537,-91473,0
C00701=34267,48132,-115518,80378,-117721,-87245,0
C00702=35169,48556,-114395,79620,-118460,-87030,0
C00703=34934,48798,-113746,79935,-118457,-86820,0
C00704=35402,49029,-113139,79550,-118851,-86705,0
C00705=35585,48842,-113640,79304,-118854,-86867,0
C00706=36145,48523,-114502,78635,-118992,-87175,0
C00707=39342,47098,-118408,74881,-119828,-88667,0
C00708=40780,47877,-116323,73699,-121108,-88284,0
C00709=36109,47981,-115956,78484,-118660,-87579,0
C00710=40181,44728,-125021,73140,-118535,-90623,0
C00711=40182,44666,-125035,73151,-118561,-90598,0
C00712=34675,44947,-124133,78983,-116158,-89720,0
C00713=36403,45653,-122187,77428,-117449,-89347,0
C00714=36332,48408,-114677,78439,-119080,-87219,0
C00715=40993,44693,-124975,72306,-118950,-90682,0
C00716=39986,44231,-126272,73202,-118138,-90922,0
C00717=35369,47938,-115920,79242,-118277,-87454,0
C00718=36254,48368,-114780,78503,-119015,-87238,0
C00719=35639,48732,-113800,79242,-118872,-86890,0
C00720=36513,49180,-112625,78531,-119622,-86667,0
C00721=42222,44651,-125120,70990,-119470,-90881,0
C00722=39854,43570,-128176,73109,-117563,-91446,0
C00723=34267,48076,-115530,80388,-117739,-87220,0
C00724=35169,48501,-114408,79631,-118477,-87006,0
C00725=34934,48743,-113759,79946,-118474,-86796,0
C00726=35402,48974,-113152,79560,-118869,-86681,0
C00727=35585,48787,-113653,79315,-118871,-86843,0
C00728=36146,48467,-114515,78646,-119010,-87151,0
C00729=39342,47041,-118420,74893,-119850,-88643,0
C00730=40747,47801,-116386,73738,-121100,-88270,0
C00731=36109,47924,-115969,78495,-118678,-87555,0
C00732=40182,44666,-125035,73151,-118561,-90598,0
C00733=40182,44605,-125048,73162,-118585,-90572,0
C00734=34714,44902,-124104,78957,-116206,-89685,0
C00735=36404,45593,-122201,77439,-117470,-89322,0
C00736=36333,48352,-114690,78450,-119100,-87195,0
C00737=40993,44632,-124988,72318,-118976,-90657,0
C00738=39987,44169,-126284,73213,-118163,-90896,0
C00739=35369,47881,-115934,79253,-118295,-87430,0
C00740=36255,48313,-114793,78514,-119033,-87215,0
C00741=35640,48676,-113813,79253,-118889,-86866,0
C00742=36513,49125,-112638,78542,-119641,-86644,0
C00743=42222,44590,-125134,71001,-119496,-90856,0
C00744=39854,43507,-128189,73120,-117588,-91420,0
C00745=34268,48019,-115543,80398,-117756,-87196,0
C00746=35170,48445,-114421,79641,-118495,-86982,0
C00747=34934,48687,-113772,79956,-118492,-86772,0
C00748=35403,48919,-113165,79571,-118886,-86656,0
C00749=35586,48731,-113666,79326,-118889,-86819,0
C00750=36146,48411,-114528,78657,-119028,-87127,0
C00751=39343,46983,-118434,74904,-119872,-88618,0
C00752=40714,47726,-116450,73778,-121092,-88254,0
C00753=36110,47868,-115982,78506,-118696,-87530,0
C00754=40182,44605,-125048,73162,-118585,-90572,0
C00755=40183,44543,-125061,73174,-118610,-90546,0
C00756=34753,44856,-124075,78931,-116254,-89651,0
C00757=36404,45533,-122214,77449,-117491,-89295,0
C00758=36333,48296,-114703,78461,-119118,-87171,0
C00759=40993,44571,-125002,72329,-119001,-90631,0
C00760=39987,44107,-126298,73224,-118188,-90870,0
C00761=35370,47825,-115946,79263,-118314,-87406,0
C00762=36255,48257,-114806,78525,-119051,-87190,0
C00763=35640,48621,-113825,79264,-118908,-86842,0
C00764=36513,49070,-112650,78554,-119659,-86620,0
C00765=42222,44528,-125146,71013,-119523,-90830,0
C00766=39855,43444,-128203,73131,-117615,-91393,0
C00767=34268,47963,-115557,80408,-117774,-87172,0
C00768=35170,48389,-114433,79652,-118512,-86958,0
C00769=34935,48632,-113785,79967,-118509,-86748,0
C00770=35403,48864,-113177,79582,-118904,-86633,0
C00771=35586,48676,-113678,79336,-118907,-86795,0
C00772=36146,48355,-114541,78668,-119047,-87103,0
C00773=39343,46925,-118447,74916,-119894,-88594,0
C00774=40681,47650,-116513,73817,-121083,-88240,0
C00775=36110,47811,-115995,78517,-118716,-87506,0
C00776=40183,44543,-125061,73174,-118610,-90546,0
C00777=40183,44482,-125074,73185,-118634,-90520,0
C00778=34793,44811,-124047,78906,-116303,-89616,0
C00779=36404,45474,-122228,77460,-117511,-89270,0
C00780=36333,48240,-114715,78472,-119136,-87147,0
C00781=40994,44509,-125014,72340,-119026,-90605,0
C00782=39988,44045,-126311,73235,-118214,-90844,0
C00783=35370,47768,-115959,79274,-118332,-87381,0
C00784=36255,48201,-114818,78536,-119071,-87166,0
C00785=35640,48566,-113838,79275,-118925,-86818,0
C00786=36514,49015,-112663,78565,-119678,-86597,0
C00787=42223,44467,-125160,71025,-119549,-90805,0
C00788=39855,43380,-128217,73142,-117640,-91366,0
C00789=34268,47907,-115569,80418,-117791,-87147,0
C00790=35170,48334,-114446,79663,-118531,-86933,0
C00791=34935,48576,-113797,79977,-118526,-86724,0
C00792=35403,48808,-113190,79592,-118922,-86609,0
C00793=35586,48621,-113691,79347,-118925,-86771,0
C00794=36147,48300,-114553,78679,-119065,-87079,0
C00795=39343,46868,-118460,74928,-119916,-88570,0
C00796=40647,47575,-116575,73856,-121075,-88225,0
C00797=36110,47755,-116007,78527,-118734,-87482,0
C00798=40183,44482,-125074,73185,-118634,-90520,0
C00799=40184,44421,-125088,73196,-118660,-90494,0
C00800=34832,44765,-124018,78880,-116351,-89582,0
C00801=36405,45414,-122240,77470,-117533,-89244,0
C00802=36334,48184,-114728,78483,-119155,-87122,0
C00803=40994,44448,-125027,72352,-119051,-90580,0
C00804=39988,43983,-126324,73246,-118239,-90818,0
C00805=35370,47712,-115972,79284,-118350,-87357,0
C00806=36256,48145,-114831,78547,-119089,-87142,0
C00807=35641,48510,-113850,79285,-118943,-86794,0
C00808=36514,48960,-112676,78576,-119696,-86573,0
C00809=42223,44406,-125173,71037,-119575,-90779,0
C00810=39856,43317,-128230,73153,-117665,-91340,0
C00811=34269,47851,-115581,80428,-117808,-87122,0
C00812=35171,48278,-114459,79673,-118548,-86909,0
C00813=34935,48521,-113810,79988,-118545,-86700,0
C00814=35404,48753,-113203,79603,-118939,-86585,0
C00815=35587,48565,-113703,79358,-118942,-86747,0
C00816=36147,48244,-114566,78690,-119084,-87055,0
C00817=39344,46810,-118472,74939,-119939,-88545,0
C00818=40614,47499,-116638,73895,-121067,-88210,0
C00819=36111,47699,-116020,78538,-118754,-87457,0
C00820=40184,44421,-125088,73196,-118660,-90494,0
C00821=40184,44360,-125101,73208,-118685,-90469,0
C00822=34871,44720,-123988,78855,-116400,-89548,0
C00823=36405,45355,-122253,77481,-117554,-89218,0
C00824=36334,48129,-114740,78494,-119174,-87099,0
C00825=40995,44387,-125041,72364,-119078,-90554,0
C00826=39988,43921,-126337,73258,-118264,-90791,0
C00827=35371,47656,-115984,79295,-118369,-87332,0
C00828=36256,48089,-114843,78558,-119108,-87118,0
C00829=35641,48455,-113863,79296,-118962,-86770,0
C00830=36515,48905,-112688,78587,-119713,-86549,0
C00831=42224,44344,-125186,71049,-119602,-90754,0
C00832=39856,43254,-128243,73164,-117692,-91313,0
C00833=34269,47795,-115594,80439,-117826,-87098,0
C00834=35171,48222,-114471,79684,-118566,-86885,0
C00835=34936,48466,-113822,79998,-118562,-86676,0
C00836=35404,48698,-113215,79614,-118957,-86561,0
C00837=35587,48510,-113716,79369,-118961,-86723,0
C00838=36147,48188,-114578,78701,-119102,-87031,0
C00839=39344,46753,-118485,74951,-119960,-88520,0
C00840=40581,47424,-116701,73934,-121059,-88195,0
C00841=36111,47642,-116033,78549,-118772,-87433,0
C00842=40184,44360,-125101,73208,-118685,-90469,0
C00843=40184,44299,-125113,73219,-118709,-90443,0
C00844=34910,44675,-123959,78830,-116449,-89513,0
C00845=36405,45295,-122266,77491,-117575,-89193,0
C00846=36334,48073,-114752,78505,-119193,-87074,0
C00847=40995,44326,-125053,72375,-119103,-90528,0
C00848=39989,43859,-126350,73269,-118289,-90765,0
C00849=35371,47599,-115996,79306,-118387,-87308,0
C00850=36256,48033,-114856,78569,-119126,-87093,0
C00851=35641,48399,-113875,79307,-118979,-86746,0
C00852=36515,48851,-112700,78598,-119732,-86525,0
C00853=42224,44283,-125199,71061,-119628,-90728,0
C00854=39856,43191,-128256,73175,-117717,-91286,0
C00855=34269,47739,-115606,80449,-117844,-87074,0
C00856=35171,48167,-114483,79694,-118584,-86861,0
C00857=34936,48410,-113834,80009,-118579,-86652,0
C00858=35404,48643,-113227,79625,-118974,-86537,0
C00859=35587,48455,-113728,79380,-118979,-86699,0
C00860=36148,48133,-114590,78712,-119120,-87006,0
C00861=39344,46695,-118497,74963,-119982,-88496,0
C00862=40548,47348,-116763,73974,-121051,-88180,0
C00863=36111,47586,-116045,78560,-118792,-87408,0
C00864=40184,44299,-125113,73219,-118709,-90443,0
C00865=40185,44237,-125126,73230,-118734,-90417,0
C00866=34949,44630,-123930,78804,-116497,-89479,0
C00867=36406,45236,-122278,77502,-117595,-89167,0
C00868=36335,48017,-114765,78516,-119211,-87050,0
C00869=40996,44265,-125066,72387,-119128,-90502,0
C00870=39989,43797,-126363,73280,-118315,-90739,0
C00871=35371,47543,-116008,79316,-118406,-87283,0
C00872=36257,47978,-114868,78580,-119146,-87070,0
C00873=35642,48344,-113887,79318,-118997,-86722,0
C00874=36515,48796,-112712,78610,-119750,-86502,0
C00875=42225,44222,-125212,71073,-119655,-90703,0
C00876=39857,43128,-128269,73186,-117744,-91260,0
C00877=34270,47682,-115619,80459,-117861,-87049,0
C00878=35172,48111,-114496,79705,-118602,-86836,0
C00879=34936,48355,-113847,80020,-118596,-86628,0
C00880=35405,48588,-113239,79636,-118992,-86513,0
C00881=35587,48399,-113740,79390,-118996,-86674,0
C00882=36148,48077,-114603,78723,-119140,-86983,0
C00883=39345,46638,-118510,74974,-120004,-88471,0
C00884=40515,47272,-116825,74013,-121043,-88165,0
C00885=36112,47530,-116057,78571,-118810,-87384,0
C00886=40185,44237,-125126,73230,-118734,-90417,0
C00887=40185,44176,-125138,73242,-118759,-90390,0
C00888=34988,44585,-123901,78780,-116546,-89445,0
C00889=36406,45176,-122291,77512,-117617,-89141,0
C00890=36335,47961,-114777,78527,-119231,-87026,0
C00891=40996,44204,-125079,72399,-119154,-90476,0
C00892=39990,43735,-126376,73291,-118340,-90713,0
C00893=35372,47487,-116021,79327,-118424,-87259,0
C00894=36257,47922,-114880,78591,-119164,-87045,0
C00895=35642,48289,-113899,79329,-119016,-86698,0
C00896=36516,48741,-112725,78621,-119768,-86478,0
C00897=42225,44161,-125225,71084,-119682,-90677,0
C00898=39857,43064,-128283,73197,-117769,-91232,0
C00899=34270,47626,-115630,80469,-117878,-87024,0
C00900=35172,48056,-114508,79716,-118619,-86812,0
C00901=34937,48300,-113859,80030,-118615,-86604,0
C00902=35405,48533,-113252,79646,-119010,-86489,0
C00903=35588,48344,-113753,79401,-119015,-86651,0
C00904=36148,48021,-114615,78734,-119158,-86958,0
C00905=39345,46580,-118522,74986,-120026,-88447,0
C00906=40482,47197,-116888,74053,-121035,-88150,0
C00907=36112,47473,-116069,78582,-118830,-87359,0
C00908=40185,44176,-125138,73242,-118759,-90390,0
C00909=40186,44115,-125151,73253,-118785,-90365,0
C00910=35027,44540,-123871,78755,-116594,-89410,0
C00911=36406,45117,-122303,77523,-117638,-89115,0
C00912=36335,47906,-114789,78538,-119249,-87002,0
C00913=40996,44142,-125091,72410,-119180,-90451,0
C00914=39990,43673,-126389,73303,-118365,-90686,0
C00915=35372,47431,-116033,79338,-118442,-87234,0
C00916=36257,47866,-114892,78602,-119182,-87021,0
C00917=35642,48234,-113912,79340,-119034,-86674,0
C00918=36516,48686,-112737,78632,-119787,-86454,0
C00919=42225,44099,-125237,71097,-119709,-90652,0
C00920=39858,43001,-128295,73208,-117795,-91206,0
C00921=34270,47570,-115643,80480,-117895,-87000,0
C00922=35172,48000,-114520,79726,-118638,-86788,0
C00923=34937,48245,-113871,80041,-118632,-86579,0
C00924=35405,48478,-113264,79657,-119027,-86465,0
C00925=35588,48289,-113765,79412,-119032,-86626,0
C00926=36149,47966,-114627,78745,-119177,-86934,0
C00927=39346,46523,-118534,74998,-120048,-88422,0
C00928=40448,47121,-116951,74092,-121026,-88135,0
C00929=36112,47417,-116081,78593,-118848,-87335,0
C00930=40186,44115,-125151,73253,-118785,-90365,0
C00931=40186,44054,-125164,73265,-118809,-90339,0
C00932=35066,44495,-123841,78730,-116644,-89376,0
C00933=36407,45057,-122315,77534,-117659,-89090,0
C00934=36336,47850,-114801,78549,-119267,-86977,0
C00935=40997,44081,-125104,72422,-119205,-90425,0
C00936=39990,43611,-126401,73314,-118391,-90660,0
C00937=35372,47374,-116045,79348,-118461,-87209,0
C00938=36258,47811,-114904,78613,-119202,-86996,0
C00939=35643,48178,-113924,79351,-119051,-86649,0
C00940=36516,48632,-112749,78644,-119805,-86430,0
C00941=42226,44038,-125250,71109,-119735,-90625,0
C00942=39858,42938,-128308,73219,-117821,-91179,0
C00943=34271,47514,-115656,80490,-117914,-86975,0
C00944=35173,47945,-114532,79737,-118656,-86764,0
C00945=34937,48189,-113883,80052,-118649,-86555,0
C00946=35406,48423,-113276,79668,-119046,-86441,0
//INST
///DATE 2025/02/20 16:20
///COMM Generated using RoboDK
///ATTR SC,RW
///GROUP1 RB1
NOP
MOVL C00000 V=30.0 PL=1
MOVL C00001 V=30.0 PL=1
MOVL C00002 V=30.0 PL=1
MOVL C00003 V=30.0 PL=1
MOVL C00004 V=30.0 PL=1
MOVL C00005 V=30.0 PL=1
MOVL C00006 V=30.0 PL=1
MOVL C00007 V=30.0 PL=1
MOVL C00008 V=130.0 PL=1
MOVL C00009 V=130.0 PL=1
MOVL C00010 V=30.0 PL=1
MOVL C00011 V=130.0 PL=1
MOVL C00012 V=30.0 PL=1
MOVL C00013 V=130.0 PL=1
MOVL C00014 V=30.0 PL=1
MOVL C00015 V=130.0 PL=1
MOVL C00016 V=20.0 PL=1
MOVL C00017 V=130.0 PL=1
MOVL C00018 V=130.0 PL=1
MOVL C00019 V=30.0 PL=1
MOVL C00020 V=130.0 PL=1
MOVL C00021 V=60.0 PL=1
MOVL C00022 V=60.0 PL=1
MOVL C00023 V=60.0 PL=1
MOVL C00024 V=60.0 PL=1
MOVL C00025 V=130.0 PL=1
MOVL C00026 V=30.0 PL=1
MOVL C00027 V=30.0 PL=1
MOVL C00028 V=30.0 PL=1
MOVL C00029 V=30.0 PL=1
MOVL C00030 V=30.0 PL=1
MOVL C00031 V=30.0 PL=1
MOVL C00032 V=30.0 PL=1
MOVL C00033 V=30.0 PL=1
MOVL C00034 V=130.0 PL=1
MOVL C00035 V=130.0 PL=1
MOVL C00036 V=30.0 PL=1
MOVL C00037 V=130.0 PL=1
MOVL C00038 V=30.0 PL=1
MOVL C00039 V=130.0 PL=1
MOVL C00040 V=30.0 PL=1
MOVL C00041 V=130.0 PL=1
MOVL C00042 V=20.0 PL=1
MOVL C00043 V=130.0 PL=1
MOVL C00044 V=130.0 PL=1
MOVL C00045 V=30.0 PL=1
MOVL C00046 V=130.0 PL=1
MOVL C00047 V=60.0 PL=1
MOVL C00048 V=60.0 PL=1
MOVL C00049 V=60.0 PL=1
MOVL C00050 V=60.0 PL=1
MOVL C00051 V=130.0 PL=1
MOVL C00052 V=30.0 PL=1
MOVL C00053 V=30.0 PL=1
MOVL C00054 V=30.0 PL=1
MOVL C00055 V=30.0 PL=1
MOVL C00056 V=30.0 PL=1
MOVL C00057 V=30.0 PL=1
MOVL C00058 V=30.0 PL=1
MOVL C00059 V=30.0 PL=1
MOVL C00060 V=130.0 PL=1
MOVL C00061 V=130.0 PL=1
MOVL C00062 V=30.0 PL=1
MOVL C00063 V=130.0 PL=1
MOVL C00064 V=30.0 PL=1
MOVL C00065 V=130.0 PL=1
MOVL C00066 V=30.0 PL=1
MOVL C00067 V=130.0 PL=1
MOVL C00068 V=20.0 PL=1
MOVL C00069 V=130.0 PL=1
MOVL C00070 V=130.0 PL=1
MOVL C00071 V=30.0 PL=1
MOVL C00072 V=130.0 PL=1
MOVL C00073 V=60.0 PL=1
MOVL C00074 V=60.0 PL=1
MOVL C00075 V=60.0 PL=1
MOVL C00076 V=60.0 PL=1
MOVL C00077 V=130.0 PL=1
MOVL C00078 V=30.0 PL=1
MOVL C00079 V=30.0 PL=1
MOVL C00080 V=30.0 PL=1
MOVL C00081 V=30.0 PL=1
MOVL C00082 V=30.0 PL=1
MOVL C00083 V=30.0 PL=1
MOVL C00084 V=30.0 PL=1
MOVL C00085 V=30.0 PL=1
MOVL C00086 V=130.0 PL=1
MOVL C00087 V=130.0 PL=1
MOVL C00088 V=30.0 PL=1
MOVL C00089 V=130.0 PL=1
MOVL C00090 V=30.0 PL=1
MOVL C00091 V=130.0 PL=1
MOVL C00092 V=30.0 PL=1
MOVL C00093 V=130.0 PL=1
MOVL C00094 V=20.0 PL=1
MOVL C00095 V=130.0 PL=1
MOVL C00096 V=130.0 PL=1
MOVL C00097 V=30.0 PL=1
MOVL C00098 V=130.0 PL=1
MOVL C00099 V=60.0 PL=1
MOVL C00100 V=60.0 PL=1
MOVL C00101 V=60.0 PL=1
MOVL C00102 V=60.0 PL=1
MOVL C00103 V=130.0 PL=1
MOVL C00104 V=30.0 PL=1
MOVL C00105 V=30.0 PL=1
MOVL C00106 V=30.0 PL=1
MOVL C00107 V=30.0 PL=1
MOVL C00108 V=30.0 PL=1
MOVL C00109 V=30.0 PL=1
MOVL C00110 V=30.0 PL=1
MOVL C00111 V=30.0 PL=1
MOVL C00112 V=130.0 PL=1
MOVL C00113 V=130.0 PL=1
MOVL C00114 V=30.0 PL=1
MOVL C00115 V=130.0 PL=1
MOVL C00116 V=30.0 PL=1
MOVL C00117 V=130.0 PL=1
MOVL C00118 V=30.0 PL=1
MOVL C00119 V=130.0 PL=1
MOVL C00120 V=20.0 PL=1
MOVL C00121 V=130.0 PL=1
MOVL C00122 V=130.0 PL=1
MOVL C00123 V=30.0 PL=1
MOVL C00124 V=130.0 PL=1
MOVL C00125 V=60.0 PL=1
MOVL C00126 V=60.0 PL=1
MOVL C00127 V=60.0 PL=1
MOVL C00128 V=60.0 PL=1
MOVL C00129 V=130.0 PL=1
MOVL C00130 V=30.0 PL=1
MOVL C00131 V=30.0 PL=1
MOVL C00132 V=30.0 PL=1
MOVL C00133 V=30.0 PL=1
MOVL C00134 V=30.0 PL=1
MOVL C00135 V=30.0 PL=1
MOVL C00136 V=30.0 PL=1
MOVL C00137 V=30.0 PL=1
MOVL C00138 V=130.0 PL=1
MOVL C00139 V=130.0 PL=1
MOVL C00140 V=30.0 PL=1
MOVL C00141 V=130.0 PL=1
MOVL C00142 V=30.0 PL=1
MOVL C00143 V=130.0 PL=1
MOVL C00144 V=30.0 PL=1
MOVL C00145 V=130.0 PL=1
MOVL C00146 V=20.0 PL=1
MOVL C00147 V=130.0 PL=1
MOVL C00148 V=130.0 PL=1
MOVL C00149 V=30.0 PL=1
MOVL C00150 V=130.0 PL=1
MOVL C00151 V=60.0 PL=1
MOVL C00152 V=60.0 PL=1
MOVL C00153 V=60.0 PL=1
MOVL C00154 V=60.0 PL=1
MOVL C00155 V=130.0 PL=1
MOVL C00156 V=30.0 PL=1
MOVL C00157 V=30.0 PL=1
MOVL C00158 V=30.0 PL=1
MOVL C00159 V=30.0 PL=1
MOVL C00160 V=30.0 PL=1
MOVL C00161 V=30.0 PL=1
MOVL C00162 V=30.0 PL=1
MOVL C00163 V=30.0 PL=1
MOVL C00164 V=130.0 PL=1
MOVL C00165 V=130.0 PL=1
MOVL C00166 V=30.0 PL=1
MOVL C00167 V=130.0 PL=1
MOVL C00168 V=30.0 PL=1
MOVL C00169 V=130.0 PL=1
MOVL C00170 V=30.0 PL=1
MOVL C00171 V=130.0 PL=1
MOVL C00172 V=20.0 PL=1
MOVL C00173 V=130.0 PL=1
MOVL C00174 V=130.0 PL=1
MOVL C00175 V=30.0 PL=1
MOVL C00176 V=130.0 PL=1
MOVL C00177 V=60.0 PL=1
MOVL C00178 V=60.0 PL=1
MOVL C00179 V=60.0 PL=1
MOVL C00180 V=60.0 PL=1
MOVL C00181 V=130.0 PL=1
MOVL C00182 V=30.0 PL=1
MOVL C00183 V=30.0 PL=1
MOVL C00184 V=30.0 PL=1
MOVL C00185 V=30.0 PL=1
MOVL C00186 V=30.0 PL=1
MOVL C00187 V=30.0 PL=1
MOVL C00188 V=30.0 PL=1
MOVL C00189 V=30.0 PL=1
MOVL C00190 V=130.0 PL=1
MOVL C00191 V=130.0 PL=1
MOVL C00192 V=30.0 PL=1
MOVL C00193 V=130.0 PL=1
MOVL C00194 V=30.0 PL=1
MOVL C00195 V=130.0 PL=1
MOVL C00196 V=30.0 PL=1
MOVL C00197 V=130.0 PL=1
MOVL C00198 V=20.0 PL=1
MOVL C00199 V=130.0 PL=1
MOVL C00200 V=130.0 PL=1
MOVL C00201 V=30.0 PL=1
MOVL C00202 V=130.0 PL=1
MOVL C00203 V=60.0 PL=1
MOVL C00204 V=60.0 PL=1
MOVL C00205 V=60.0 PL=1
MOVL C00206 V=60.0 PL=1
MOVL C00207 V=130.0 PL=1
MOVL C00208 V=30.0 PL=1
MOVL C00209 V=30.0 PL=1
MOVL C00210 V=30.0 PL=1
MOVL C00211 V=30.0 PL=1
MOVL C00212 V=30.0 PL=1
MOVL C00213 V=30.0 PL=1
MOVL C00214 V=30.0 PL=1
MOVL C00215 V=30.0 PL=1
MOVL C00216 V=130.0 PL=1
MOVL C00217 V=130.0 PL=1
MOVL C00218 V=30.0 PL=1
MOVL C00219 V=130.0 PL=1
MOVL C00220 V=30.0 PL=1
MOVL C00221 V=130.0 PL=1
MOVL C00222 V=30.0 PL=1
MOVL C00223 V=130.0 PL=1
MOVL C00224 V=20.0 PL=1
MOVL C00225 V=130.0 PL=1
MOVL C00226 V=130.0 PL=1
MOVL C00227 V=30.0 PL=1
MOVL C00228 V=130.0 PL=1
MOVL C00229 V=60.0 PL=1
MOVL C00230 V=60.0 PL=1
MOVL C00231 V=60.0 PL=1
MOVL C00232 V=60.0 PL=1
MOVL C00233 V=130.0 PL=1
MOVL C00234 V=30.0 PL=1
MOVL C00235 V=30.0 PL=1
MOVL C00236 V=30.0 PL=1
MOVL C00237 V=30.0 PL=1
MOVL C00238 V=30.0 PL=1
MOVL C00239 V=30.0 PL=1
MOVL C00240 V=30.0 PL=1
MOVL C00241 V=30.0 PL=1
MOVL C00242 V=130.0 PL=1
MOVL C00243 V=130.0 PL=1
MOVL C00244 V=30.0 PL=1
MOVL C00245 V=130.0 PL=1
MOVL C00246 V=30.0 PL=1
MOVL C00247 V=130.0 PL=1
MOVL C00248 V=30.0 PL=1
MOVL C00249 V=130.0 PL=1
MOVL C00250 V=20.0 PL=1
MOVL C00251 V=130.0 PL=1
MOVL C00252 V=130.0 PL=1
MOVL C00253 V=30.0 PL=1
MOVL C00254 V=130.0 PL=1
MOVL C00255 V=60.0 PL=1
MOVL C00256 V=60.0 PL=1
MOVL C00257 V=60.0 PL=1
MOVL C00258 V=60.0 PL=1
MOVL C00259 V=130.0 PL=1
MOVL C00260 V=30.0 PL=1
MOVL C00261 V=30.0 PL=1
MOVL C00262 V=30.0 PL=1
MOVL C00263 V=30.0 PL=1
MOVL C00264 V=30.0 PL=1
MOVL C00265 V=30.0 PL=1
MOVL C00266 V=30.0 PL=1
MOVL C00267 V=30.0 PL=1
MOVL C00268 V=130.0 PL=1
MOVL C00269 V=130.0 PL=1
MOVL C00270 V=30.0 PL=1
MOVL C00271 V=130.0 PL=1
MOVL C00272 V=30.0 PL=1
MOVL C00273 V=130.0 PL=1
MOVL C00274 V=30.0 PL=1
MOVL C00275 V=130.0 PL=1
MOVL C00276 V=20.0 PL=1
MOVL C00277 V=130.0 PL=1
MOVL C00278 V=130.0 PL=1
MOVL C00279 V=30.0 PL=1
MOVL C00280 V=130.0 PL=1
MOVL C00281 V=60.0 PL=1
MOVL C00282 V=60.0 PL=1
MOVL C00283 V=60.0 PL=1
MOVL C00284 V=60.0 PL=1
MOVL C00285 V=130.0 PL=1
MOVL C00286 V=30.0 PL=1
MOVL C00287 V=30.0 PL=1
MOVL C00288 V=30.0 PL=1
MOVL C00289 V=30.0 PL=1
MOVL C00290 V=30.0 PL=1
MOVL C00291 V=30.0 PL=1
MOVL C00292 V=30.0 PL=1
MOVL C00293 V=30.0 PL=1
MOVL C00294 V=130.0 PL=1
MOVL C00295 V=130.0 PL=1
MOVL C00296 V=30.0 PL=1
MOVL C00297 V=130.0 PL=1
MOVL C00298 V=30.0 PL=1
MOVL C00299 V=130.0 PL=1
MOVL C00300 V=30.0 PL=1
MOVL C00301 V=130.0 PL=1
MOVL C00302 V=20.0 PL=1
MOVL C00303 V=130.0 PL=1
MOVL C00304 V=130.0 PL=1
MOVL C00305 V=30.0 PL=1
MOVL C00306 V=130.0 PL=1
MOVL C00307 V=60.0 PL=1
MOVL C00308 V=60.0 PL=1
MOVL C00309 V=60.0 PL=1
MOVL C00310 V=60.0 PL=1
MOVL C00311 V=130.0 PL=1
MOVL C00312 V=30.0 PL=1
MOVL C00313 V=30.0 PL=1
MOVL C00314 V=30.0 PL=1
MOVL C00315 V=30.0 PL=1
MOVL C00316 V=30.0 PL=1
MOVL C00317 V=30.0 PL=1
MOVL C00318 V=30.0 PL=1
MOVL C00319 V=30.0 PL=1
MOVL C00320 V=130.0 PL=1
MOVL C00321 V=130.0 PL=1
MOVL C00322 V=30.0 PL=1
MOVL C00323 V=130.0 PL=1
MOVL C00324 V=30.0 PL=1
MOVL C00325 V=130.0 PL=1
MOVL C00326 V=30.0 PL=1
MOVL C00327 V=130.0 PL=1
MOVL C00328 V=20.0 PL=1
MOVL C00329 V=130.0 PL=1
MOVL C00330 V=130.0 PL=1
MOVL C00331 V=30.0 PL=1
MOVL C00332 V=130.0 PL=1
MOVL C00333 V=60.0 PL=1
MOVL C00334 V=60.0 PL=1
MOVL C00335 V=60.0 PL=1
MOVL C00336 V=60.0 PL=1
MOVL C00337 V=130.0 PL=1
MOVL C00338 V=30.0 PL=1
MOVL C00339 V=30.0 PL=1
MOVL C00340 V=30.0 PL=1
MOVL C00341 V=30.0 PL=1
MOVL C00342 V=30.0 PL=1
MOVL C00343 V=30.0 PL=1
MOVL C00344 V=30.0 PL=1
MOVL C00345 V=30.0 PL=1
MOVL C00346 V=130.0 PL=1
MOVL C00347 V=130.0 PL=1
MOVL C00348 V=30.0 PL=1
MOVL C00349 V=130.0 PL=1
MOVL C00350 V=30.0 PL=1
MOVL C00351 V=130.0 PL=1
MOVL C00352 V=30.0 PL=1
MOVL C00353 V=130.0 PL=1
MOVL C00354 V=20.0 PL=1
MOVL C00355 V=130.0 PL=1
MOVL C00356 V=130.0 PL=1
MOVL C00357 V=30.0 PL=1
MOVL C00358 V=130.0 PL=1
MOVL C00359 V=60.0 PL=1
MOVL C00360 V=60.0 PL=1
MOVL C00361 V=60.0 PL=1
MOVL C00362 V=60.0 PL=1
MOVL C00363 V=130.0 PL=1
MOVL C00364 V=30.0 PL=1
MOVL C00365 V=30.0 PL=1
MOVL C00366 V=30.0 PL=1
MOVL C00367 V=30.0 PL=1
MOVL C00368 V=30.0 PL=1
MOVL C00369 V=30.0 PL=1
MOVL C00370 V=30.0 PL=1
MOVL C00371 V=30.0 PL=1
MOVL C00372 V=130.0 PL=1
MOVL C00373 V=130.0 PL=1
MOVL C00374 V=30.0 PL=1
MOVL C00375 V=130.0 PL=1
MOVL C00376 V=30.0 PL=1
MOVL C00377 V=130.0 PL=1
MOVL C00378 V=30.0 PL=1
MOVL C00379 V=130.0 PL=1
MOVL C00380 V=20.0 PL=1
MOVL C00381 V=130.0 PL=1
MOVL C00382 V=130.0 PL=1
MOVL C00383 V=30.0 PL=1
MOVL C00384 V=130.0 PL=1
MOVL C00385 V=60.0 PL=1
MOVL C00386 V=60.0 PL=1
MOVL C00387 V=60.0 PL=1
MOVL C00388 V=60.0 PL=1
MOVL C00389 V=130.0 PL=1
MOVL C00390 V=30.0 PL=1
MOVL C00391 V=30.0 PL=1
MOVL C00392 V=30.0 PL=1
MOVL C00393 V=30.0 PL=1
MOVL C00394 V=30.0 PL=1
MOVL C00395 V=30.0 PL=1
MOVL C00396 V=30.0 PL=1
MOVL C00397 V=30.0 PL=1
MOVL C00398 V=130.0 PL=1
MOVL C00399 V=130.0 PL=1
MOVL C00400 V=30.0 PL=1
MOVL C00401 V=130.0 PL=1
MOVL C00402 V=30.0 PL=1
MOVL C00403 V=130.0 PL=1
MOVL C00404 V=30.0 PL=1
MOVL C00405 V=130.0 PL=1
MOVL C00406 V=20.0 PL=1
MOVL C00407 V=130.0 PL=1
MOVL C00408 V=130.0 PL=1
MOVL C00409 V=30.0 PL=1
MOVL C00410 V=130.0 PL=1
MOVL C00411 V=60.0 PL=1
MOVL C00412 V=60.0 PL=1
MOVL C00413 V=60.0 PL=1
MOVL C00414 V=60.0 PL=1
MOVL C00415 V=130.0 PL=1
MOVL C00416 V=30.0 PL=1
MOVL C00417 V=30.0 PL=1
MOVL C00418 V=30.0 PL=1
MOVL C00419 V=30.0 PL=1
MOVL C00420 V=30.0 PL=1
MOVL C00421 V=30.0 PL=1
MOVL C00422 V=30.0 PL=1
MOVL C00423 V=30.0 PL=1
MOVL C00424 V=130.0 PL=1
MOVL C00425 V=130.0 PL=1
MOVL C00426 V=30.0 PL=1
MOVL C00427 V=130.0 PL=1
MOVL C00428 V=30.0 PL=1
MOVL C00429 V=130.0 PL=1
MOVL C00430 V=30.0 PL=1
MOVL C00431 V=130.0 PL=1
MOVL C00432 V=20.0 PL=1
MOVL C00433 V=130.0 PL=1
MOVL C00434 V=130.0 PL=1
MOVL C00435 V=30.0 PL=1
MOVL C00436 V=130.0 PL=1
MOVL C00437 V=60.0 PL=1
MOVL C00438 V=60.0 PL=1
MOVL C00439 V=60.0 PL=1
MOVL C00440 V=60.0 PL=1
MOVL C00441 V=130.0 PL=1
MOVL C00442 V=30.0 PL=1
MOVL C00443 V=30.0 PL=1
MOVL C00444 V=30.0 PL=1
MOVL C00445 V=30.0 PL=1
MOVL C00446 V=30.0 PL=1
MOVL C00447 V=30.0 PL=1
MOVL C00448 V=30.0 PL=1
MOVL C00449 V=30.0 PL=1
MOVL C00450 V=130.0 PL=1
MOVL C00451 V=130.0 PL=1
MOVL C00452 V=30.0 PL=1
MOVL C00453 V=130.0 PL=1
MOVL C00454 V=30.0 PL=1
MOVL C00455 V=130.0 PL=1
MOVL C00456 V=30.0 PL=1
MOVL C00457 V=130.0 PL=1
MOVL C00458 V=20.0 PL=1
MOVL C00459 V=130.0 PL=1
MOVL C00460 V=130.0 PL=1
MOVL C00461 V=30.0 PL=1
MOVL C00462 V=130.0 PL=1
MOVL C00463 V=60.0 PL=1
MOVL C00464 V=60.0 PL=1
MOVL C00465 V=60.0 PL=1
MOVL C00466 V=60.0 PL=1
MOVL C00467 V=130.0 PL=1
MOVL C00468 V=30.0 PL=1
MOVL C00469 V=30.0 PL=1
MOVL C00470 V=30.0 PL=1
MOVL C00471 V=30.0 PL=1
MOVL C00472 V=30.0 PL=1
MOVL C00473 V=30.0 PL=1
MOVL C00474 V=30.0 PL=1
MOVL C00475 V=30.0 PL=1
MOVL C00476 V=130.0 PL=1
MOVL C00477 V=130.0 PL=1
MOVL C00478 V=30.0 PL=1
MOVL C00479 V=130.0 PL=1
MOVL C00480 V=30.0 PL=1
MOVL C00481 V=130.0 PL=1
MOVL C00482 V=30.0 PL=1
MOVL C00483 V=130.0 PL=1
MOVL C00484 V=20.0 PL=1
MOVL C00485 V=130.0 PL=1
MOVL C00486 V=130.0 PL=1
MOVL C00487 V=30.0 PL=1
MOVL C00488 V=130.0 PL=1
MOVL C00489 V=60.0 PL=1
MOVL C00490 V=60.0 PL=1
MOVL C00491 V=60.0 PL=1
MOVL C00492 V=60.0 PL=1
MOVL C00493 V=130.0 PL=1
MOVL C00494 V=30.0 PL=1
MOVL C00495 V=30.0 PL=1
MOVL C00496 V=30.0 PL=1
MOVL C00497 V=30.0 PL=1
MOVL C00498 V=30.0 PL=1
MOVL C00499 V=30.0 PL=1
MOVL C00500 V=30.0 PL=1
MOVL C00501 V=30.0 PL=1
MOVL C00502 V=130.0 PL=1
MOVL C00503 V=130.0 PL=1
MOVL C00504 V=30.0 PL=1
MOVL C00505 V=130.0 PL=1
MOVL C00506 V=30.0 PL=1
MOVL C00507 V=130.0 PL=1
MOVL C00508 V=30.0 PL=1
MOVL C00509 V=130.0 PL=1
MOVL C00510 V=20.0 PL=1
MOVL C00511 V=130.0 PL=1
MOVL C00512 V=130.0 PL=1
MOVL C00513 V=30.0 PL=1
MOVL C00514 V=130.0 PL=1
MOVL C00515 V=60.0 PL=1
MOVL C00516 V=60.0 PL=1
MOVL C00517 V=60.0 PL=1
MOVL C00518 V=60.0 PL=1
MOVL C00519 V=130.0 PL=1
MOVL C00520 V=30.0 PL=1
MOVL C00521 V=30.0 PL=1
MOVL C00522 V=30.0 PL=1
MOVL C00523 V=30.0 PL=1
MOVL C00524 V=30.0 PL=1
MOVL C00525 V=30.0 PL=1
MOVL C00526 V=30.0 PL=1
MOVL C00527 V=30.0 PL=1
MOVL C00528 V=130.0 PL=1
MOVL C00529 V=130.0 PL=1
MOVL C00530 V=30.0 PL=1
MOVL C00531 V=130.0 PL=1
MOVL C00532 V=30.0 PL=1
MOVL C00533 V=130.0 PL=1
MOVL C00534 V=30.0 PL=1
MOVL C00535 V=130.0 PL=1
MOVL C00536 V=20.0 PL=1
MOVL C00537 V=130.0 PL=1
MOVL C00538 V=130.0 PL=1
MOVL C00539 V=30.0 PL=1
MOVL C00540 V=130.0 PL=1
MOVL C00541 V=60.0 PL=1
MOVL C00542 V=60.0 PL=1
MOVL C00543 V=60.0 PL=1
MOVL C00544 V=60.0 PL=1
MOVL C00545 V=130.0 PL=1
MOVL C00546 V=30.0 PL=1
MOVL C00547 V=30.0 PL=1
MOVL C00548 V=30.0 PL=1
MOVL C00549 V=30.0 PL=1
MOVL C00550 V=30.0 PL=1
MOVL C00551 V=30.0 PL=1
MOVL C00552 V=30.0 PL=1
MOVL C00553 V=30.0 PL=1
MOVL C00554 V=130.0 PL=1
MOVL C00555 V=130.0 PL=1
MOVL C00556 V=30.0 PL=1
MOVL C00557 V=130.0 PL=1
MOVL C00558 V=30.0 PL=1
MOVL C00559 V=130.0 PL=1
MOVL C00560 V=30.0 PL=1
MOVL C00561 V=130.0 PL=1
MOVL C00562 V=20.0 PL=1
MOVL C00563 V=130.0 PL=1
MOVL C00564 V=130.0 PL=1
MOVL C00565 V=30.0 PL=1
MOVL C00566 V=130.0 PL=1
MOVL C00567 V=60.0 PL=1
MOVL C00568 V=60.0 PL=1
MOVL C00569 V=60.0 PL=1
MOVL C00570 V=60.0 PL=1
MOVL C00571 V=130.0 PL=1
MOVL C00572 V=30.0 PL=1
MOVL C00573 V=30.0 PL=1
MOVL C00574 V=30.0 PL=1
MOVL C00575 V=30.0 PL=1
MOVL C00576 V=30.0 PL=1
MOVL C00577 V=30.0 PL=1
MOVL C00578 V=30.0 PL=1
MOVL C00579 V=30.0 PL=1
MOVL C00580 V=130.0 PL=1
MOVL C00581 V=130.0 PL=1
MOVL C00582 V=30.0 PL=1
MOVL C00583 V=130.0 PL=1
MOVL C00584 V=30.0 PL=1
MOVL C00585 V=130.0 PL=1
MOVL C00586 V=30.0 PL=1
MOVL C00587 V=130.0 PL=1
MOVL C00588 V=20.0 PL=1
MOVL C00589 V=130.0 PL=1
MOVL C00590 V=130.0 PL=1
MOVL C00591 V=30.0 PL=1
MOVL C00592 V=130.0 PL=1
MOVL C00593 V=60.0 PL=1
MOVL C00594 V=60.0 PL=1
MOVL C00595 V=60.0 PL=1
MOVL C00596 V=60.0 PL=1
MOVL C00597 V=130.0 PL=1
MOVL C00598 V=30.0 PL=1
MOVL C00599 V=30.0 PL=1
MOVL C00600 V=30.0 PL=1
MOVL C00601 V=30.0 PL=1
MOVL C00602 V=30.0 PL=1
MOVL C00603 V=30.0 PL=1
MOVL C00604 V=30.0 PL=1
MOVL C00605 V=30.0 PL=1
MOVL C00606 V=130.0 PL=1
MOVL C00607 V=130.0 PL=1
MOVL C00608 V=30.0 PL=1
MOVL C00609 V=130.0 PL=1
MOVL C00610 V=30.0 PL=1
MOVL C00611 V=130.0 PL=1
MOVL C00612 V=30.0 PL=1
MOVL C00613 V=130.0 PL=1
MOVL C00614 V=20.0 PL=1
MOVL C00615 V=130.0 PL=1
MOVL C00616 V=130.0 PL=1
MOVL C00617 V=30.0 PL=1
MOVL C00618 V=130.0 PL=1
MOVL C00619 V=60.0 PL=1
MOVL C00620 V=60.0 PL=1
MOVL C00621 V=60.0 PL=1
MOVL C00622 V=60.0 PL=1
MOVL C00623 V=130.0 PL=1
MOVL C00624 V=30.0 PL=1
MOVL C00625 V=30.0 PL=1
MOVL C00626 V=30.0 PL=1
MOVL C00627 V=30.0 PL=1
MOVL C00628 V=30.0 PL=1
MOVL C00629 V=30.0 PL=1
MOVL C00630 V=30.0 PL=1
MOVL C00631 V=30.0 PL=1
MOVL C00632 V=130.0 PL=1
MOVL C00633 V=130.0 PL=1
MOVL C00634 V=30.0 PL=1
MOVL C00635 V=130.0 PL=1
MOVL C00636 V=30.0 PL=1
MOVL C00637 V=130.0 PL=1
MOVL C00638 V=30.0 PL=1
MOVL C00639 V=130.0 PL=1
MOVL C00640 V=20.0 PL=1
MOVL C00641 V=130.0 PL=1
MOVL C00642 V=130.0 PL=1
MOVL C00643 V=30.0 PL=1
MOVL C00644 V=130.0 PL=1
MOVL C00645 V=60.0 PL=1
MOVL C00646 V=60.0 PL=1
MOVL C00647 V=60.0 PL=1
MOVL C00648 V=60.0 PL=1
MOVL C00649 V=130.0 PL=1
MOVL C00650 V=30.0 PL=1
MOVL C00651 V=30.0 PL=1
MOVL C00652 V=30.0 PL=1
MOVL C00653 V=30.0 PL=1
MOVL C00654 V=30.0 PL=1
MOVL C00655 V=30.0 PL=1
MOVL C00656 V=30.0 PL=1
MOVL C00657 V=30.0 PL=1
MOVL C00658 V=130.0 PL=1
MOVL C00659 V=130.0 PL=1
MOVL C00660 V=30.0 PL=1
MOVL C00661 V=130.0 PL=1
MOVL C00662 V=30.0 PL=1
MOVL C00663 V=130.0 PL=1
MOVL C00664 V=30.0 PL=1
MOVL C00665 V=130.0 PL=1
MOVL C00666 V=20.0 PL=1
MOVL C00667 V=130.0 PL=1
MOVL C00668 V=130.0 PL=1
MOVL C00669 V=30.0 PL=1
MOVL C00670 V=130.0 PL=1
MOVL C00671 V=60.0 PL=1
MOVL C00672 V=60.0 PL=1
MOVL C00673 V=60.0 PL=1
MOVL C00674 V=60.0 PL=1
MOVL C00675 V=130.0 PL=1
MOVL C00676 V=30.0 PL=1
MOVL C00677 V=30.0 PL=1
MOVL C00678 V=30.0 PL=1
MOVL C00679 V=30.0 PL=1
MOVL C00680 V=30.0 PL=1
MOVL C00681 V=30.0 PL=1
MOVL C00682 V=30.0 PL=1
MOVL C00683 V=30.0 PL=1
MOVL C00684 V=130.0 PL=1
MOVL C00685 V=130.0 PL=1
MOVL C00686 V=30.0 PL=1
MOVL C00687 V=130.0 PL=1
MOVL C00688 V=20.0 PL=1
MOVL C00689 V=130.0 PL=1
MOVL C00690 V=130.0 PL=1
MOVL C00691 V=30.0 PL=1
MOVL C00692 V=130.0 PL=1
MOVL C00693 V=60.0 PL=1
MOVL C00694 V=60.0 PL=1
MOVL C00695 V=60.0 PL=1
MOVL C00696 V=60.0 PL=1
MOVL C00697 V=130.0 PL=1
MOVL C00698 V=30.0 PL=1
MOVL C00699 V=30.0 PL=1
MOVL C00700 V=30.0 PL=1
MOVL C00701 V=30.0 PL=1
MOVL C00702 V=30.0 PL=1
MOVL C00703 V=30.0 PL=1
MOVL C00704 V=30.0 PL=1
MOVL C00705 V=30.0 PL=1
MOVL C00706 V=130.0 PL=1
MOVL C00707 V=130.0 PL=1
MOVL C00708 V=30.0 PL=1
MOVL C00709 V=130.0 PL=1
MOVL C00710 V=20.0 PL=1
MOVL C00711 V=130.0 PL=1
MOVL C00712 V=130.0 PL=1
MOVL C00713 V=30.0 PL=1
MOVL C00714 V=130.0 PL=1
MOVL C00715 V=60.0 PL=1
MOVL C00716 V=60.0 PL=1
MOVL C00717 V=60.0 PL=1
MOVL C00718 V=60.0 PL=1
MOVL C00719 V=130.0 PL=1
MOVL C00720 V=30.0 PL=1
MOVL C00721 V=30.0 PL=1
MOVL C00722 V=30.0 PL=1
MOVL C00723 V=30.0 PL=1
MOVL C00724 V=30.0 PL=1
MOVL C00725 V=30.0 PL=1
MOVL C00726 V=30.0 PL=1
MOVL C00727 V=30.0 PL=1
MOVL C00728 V=130.0 PL=1
MOVL C00729 V=130.0 PL=1
MOVL C00730 V=30.0 PL=1
MOVL C00731 V=130.0 PL=1
MOVL C00732 V=20.0 PL=1
MOVL C00733 V=130.0 PL=1
MOVL C00734 V=130.0 PL=1
MOVL C00735 V=30.0 PL=1
MOVL C00736 V=130.0 PL=1
MOVL C00737 V=60.0 PL=1
MOVL C00738 V=60.0 PL=1
MOVL C00739 V=60.0 PL=1
MOVL C00740 V=60.0 PL=1
MOVL C00741 V=130.0 PL=1
MOVL C00742 V=30.0 PL=1
MOVL C00743 V=30.0 PL=1
MOVL C00744 V=30.0 PL=1
MOVL C00745 V=30.0 PL=1
MOVL C00746 V=30.0 PL=1
MOVL C00747 V=30.0 PL=1
MOVL C00748 V=30.0 PL=1
MOVL C00749 V=30.0 PL=1
MOVL C00750 V=130.0 PL=1
MOVL C00751 V=130.0 PL=1
MOVL C00752 V=30.0 PL=1
MOVL C00753 V=130.0 PL=1
MOVL C00754 V=20.0 PL=1
MOVL C00755 V=130.0 PL=1
MOVL C00756 V=130.0 PL=1
MOVL C00757 V=30.0 PL=1
MOVL C00758 V=130.0 PL=1
MOVL C00759 V=60.0 PL=1
MOVL C00760 V=60.0 PL=1
MOVL C00761 V=60.0 PL=1
MOVL C00762 V=60.0 PL=1
MOVL C00763 V=130.0 PL=1
MOVL C00764 V=30.0 PL=1
MOVL C00765 V=30.0 PL=1
MOVL C00766 V=30.0 PL=1
MOVL C00767 V=30.0 PL=1
MOVL C00768 V=30.0 PL=1
MOVL C00769 V=30.0 PL=1
MOVL C00770 V=30.0 PL=1
MOVL C00771 V=30.0 PL=1
MOVL C00772 V=130.0 PL=1
MOVL C00773 V=130.0 PL=1
MOVL C00774 V=30.0 PL=1
MOVL C00775 V=130.0 PL=1
MOVL C00776 V=20.0 PL=1
MOVL C00777 V=130.0 PL=1
MOVL C00778 V=130.0 PL=1
MOVL C00779 V=30.0 PL=1
MOVL C00780 V=130.0 PL=1
MOVL C00781 V=60.0 PL=1
MOVL C00782 V=60.0 PL=1
MOVL C00783 V=60.0 PL=1
MOVL C00784 V=60.0 PL=1
MOVL C00785 V=130.0 PL=1
MOVL C00786 V=30.0 PL=1
MOVL C00787 V=30.0 PL=1
MOVL C00788 V=30.0 PL=1
MOVL C00789 V=30.0 PL=1
MOVL C00790 V=30.0 PL=1
MOVL C00791 V=30.0 PL=1
MOVL C00792 V=30.0 PL=1
MOVL C00793 V=30.0 PL=1
MOVL C00794 V=130.0 PL=1
MOVL C00795 V=130.0 PL=1
MOVL C00796 V=30.0 PL=1
MOVL C00797 V=130.0 PL=1
MOVL C00798 V=20.0 PL=1
MOVL C00799 V=130.0 PL=1
MOVL C00800 V=130.0 PL=1
MOVL C00801 V=30.0 PL=1
MOVL C00802 V=130.0 PL=1
MOVL C00803 V=60.0 PL=1
MOVL C00804 V=60.0 PL=1
MOVL C00805 V=60.0 PL=1
MOVL C00806 V=60.0 PL=1
MOVL C00807 V=130.0 PL=1
MOVL C00808 V=30.0 PL=1
MOVL C00809 V=30.0 PL=1
MOVL C00810 V=30.0 PL=1
MOVL C00811 V=30.0 PL=1
MOVL C00812 V=30.0 PL=1
MOVL C00813 V=30.0 PL=1
MOVL C00814 V=30.0 PL=1
MOVL C00815 V=30.0 PL=1
MOVL C00816 V=130.0 PL=1
MOVL C00817 V=130.0 PL=1
MOVL C00818 V=30.0 PL=1
MOVL C00819 V=130.0 PL=1
MOVL C00820 V=20.0 PL=1
MOVL C00821 V=130.0 PL=1
MOVL C00822 V=130.0 PL=1
MOVL C00823 V=30.0 PL=1
MOVL C00824 V=130.0 PL=1
MOVL C00825 V=60.0 PL=1
MOVL C00826 V=60.0 PL=1
MOVL C00827 V=60.0 PL=1
MOVL C00828 V=60.0 PL=1
MOVL C00829 V=130.0 PL=1
MOVL C00830 V=30.0 PL=1
MOVL C00831 V=30.0 PL=1
MOVL C00832 V=30.0 PL=1
MOVL C00833 V=30.0 PL=1
MOVL C00834 V=30.0 PL=1
MOVL C00835 V=30.0 PL=1
MOVL C00836 V=30.0 PL=1
MOVL C00837 V=30.0 PL=1
MOVL C00838 V=130.0 PL=1
MOVL C00839 V=130.0 PL=1
MOVL C00840 V=30.0 PL=1
MOVL C00841 V=130.0 PL=1
MOVL C00842 V=20.0 PL=1
MOVL C00843 V=130.0 PL=1
MOVL C00844 V=130.0 PL=1
MOVL C00845 V=30.0 PL=1
MOVL C00846 V=130.0 PL=1
MOVL C00847 V=60.0 PL=1
MOVL C00848 V=60.0 PL=1
MOVL C00849 V=60.0 PL=1
MOVL C00850 V=60.0 PL=1
MOVL C00851 V=130.0 PL=1
MOVL C00852 V=30.0 PL=1
MOVL C00853 V=30.0 PL=1
MOVL C00854 V=30.0 PL=1
MOVL C00855 V=30.0 PL=1
MOVL C00856 V=30.0 PL=1
MOVL C00857 V=30.0 PL=1
MOVL C00858 V=30.0 PL=1
MOVL C00859 V=30.0 PL=1
MOVL C00860 V=130.0 PL=1
MOVL C00861 V=130.0 PL=1
MOVL C00862 V=30.0 PL=1
MOVL C00863 V=130.0 PL=1
MOVL C00864 V=20.0 PL=1
MOVL C00865 V=130.0 PL=1
MOVL C00866 V=130.0 PL=1
MOVL C00867 V=30.0 PL=1
MOVL C00868 V=130.0 PL=1
MOVL C00869 V=60.0 PL=1
MOVL C00870 V=60.0 PL=1
MOVL C00871 V=60.0 PL=1
MOVL C00872 V=60.0 PL=1
MOVL C00873 V=130.0 PL=1
MOVL C00874 V=30.0 PL=1
MOVL C00875 V=30.0 PL=1
MOVL C00876 V=30.0 PL=1
MOVL C00877 V=30.0 PL=1
MOVL C00878 V=30.0 PL=1
MOVL C00879 V=30.0 PL=1
MOVL C00880 V=30.0 PL=1
MOVL C00881 V=30.0 PL=1
MOVL C00882 V=130.0 PL=1
MOVL C00883 V=130.0 PL=1
MOVL C00884 V=30.0 PL=1
MOVL C00885 V=130.0 PL=1
MOVL C00886 V=20.0 PL=1
MOVL C00887 V=130.0 PL=1
MOVL C00888 V=130.0 PL=1
MOVL C00889 V=30.0 PL=1
MOVL C00890 V=130.0 PL=1
MOVL C00891 V=60.0 PL=1
MOVL C00892 V=60.0 PL=1
MOVL C00893 V=60.0 PL=1
MOVL C00894 V=60.0 PL=1
MOVL C00895 V=130.0 PL=1
MOVL C00896 V=30.0 PL=1
MOVL C00897 V=30.0 PL=1
MOVL C00898 V=30.0 PL=1
MOVL C00899 V=30.0 PL=1
MOVL C00900 V=30.0 PL=1
MOVL C00901 V=30.0 PL=1
MOVL C00902 V=30.0 PL=1
MOVL C00903 V=30.0 PL=1
MOVL C00904 V=130.0 PL=1
MOVL C00905 V=130.0 PL=1
MOVL C00906 V=30.0 PL=1
MOVL C00907 V=130.0 PL=1
MOVL C00908 V=20.0 PL=1
MOVL C00909 V=130.0 PL=1
MOVL C00910 V=130.0 PL=1
MOVL C00911 V=30.0 PL=1
MOVL C00912 V=130.0 PL=1
MOVL C00913 V=60.0 PL=1
MOVL C00914 V=60.0 PL=1
MOVL C00915 V=60.0 PL=1
MOVL C00916 V=60.0 PL=1
MOVL C00917 V=130.0 PL=1
MOVL C00918 V=30.0 PL=1
MOVL C00919 V=30.0 PL=1
MOVL C00920 V=30.0 PL=1
MOVL C00921 V=30.0 PL=1
MOVL C00922 V=30.0 PL=1
MOVL C00923 V=30.0 PL=1
MOVL C00924 V=30.0 PL=1
MOVL C00925 V=30.0 PL=1
MOVL C00926 V=130.0 PL=1
MOVL C00927 V=130.0 PL=1
MOVL C00928 V=30.0 PL=1
MOVL C00929 V=130.0 PL=1
MOVL C00930 V=20.0 PL=1
MOVL C00931 V=130.0 PL=1
MOVL C00932 V=130.0 PL=1
MOVL C00933 V=30.0 PL=1
MOVL C00934 V=130.0 PL=1
MOVL C00935 V=60.0 PL=1
MOVL C00936 V=60.0 PL=1
MOVL C00937 V=60.0 PL=1
MOVL C00938 V=60.0 PL=1
MOVL C00939 V=130.0 PL=1
MOVL C00940 V=30.0 PL=1
MOVL C00941 V=30.0 PL=1
MOVL C00942 V=30.0 PL=1
MOVL C00943 V=30.0 PL=1
MOVL C00944 V=30.0 PL=1
MOVL C00945 V=30.0 PL=1
MOVL C00946 V=30.0 PL=1
END
